REGION Network 49: Main Op Local Control
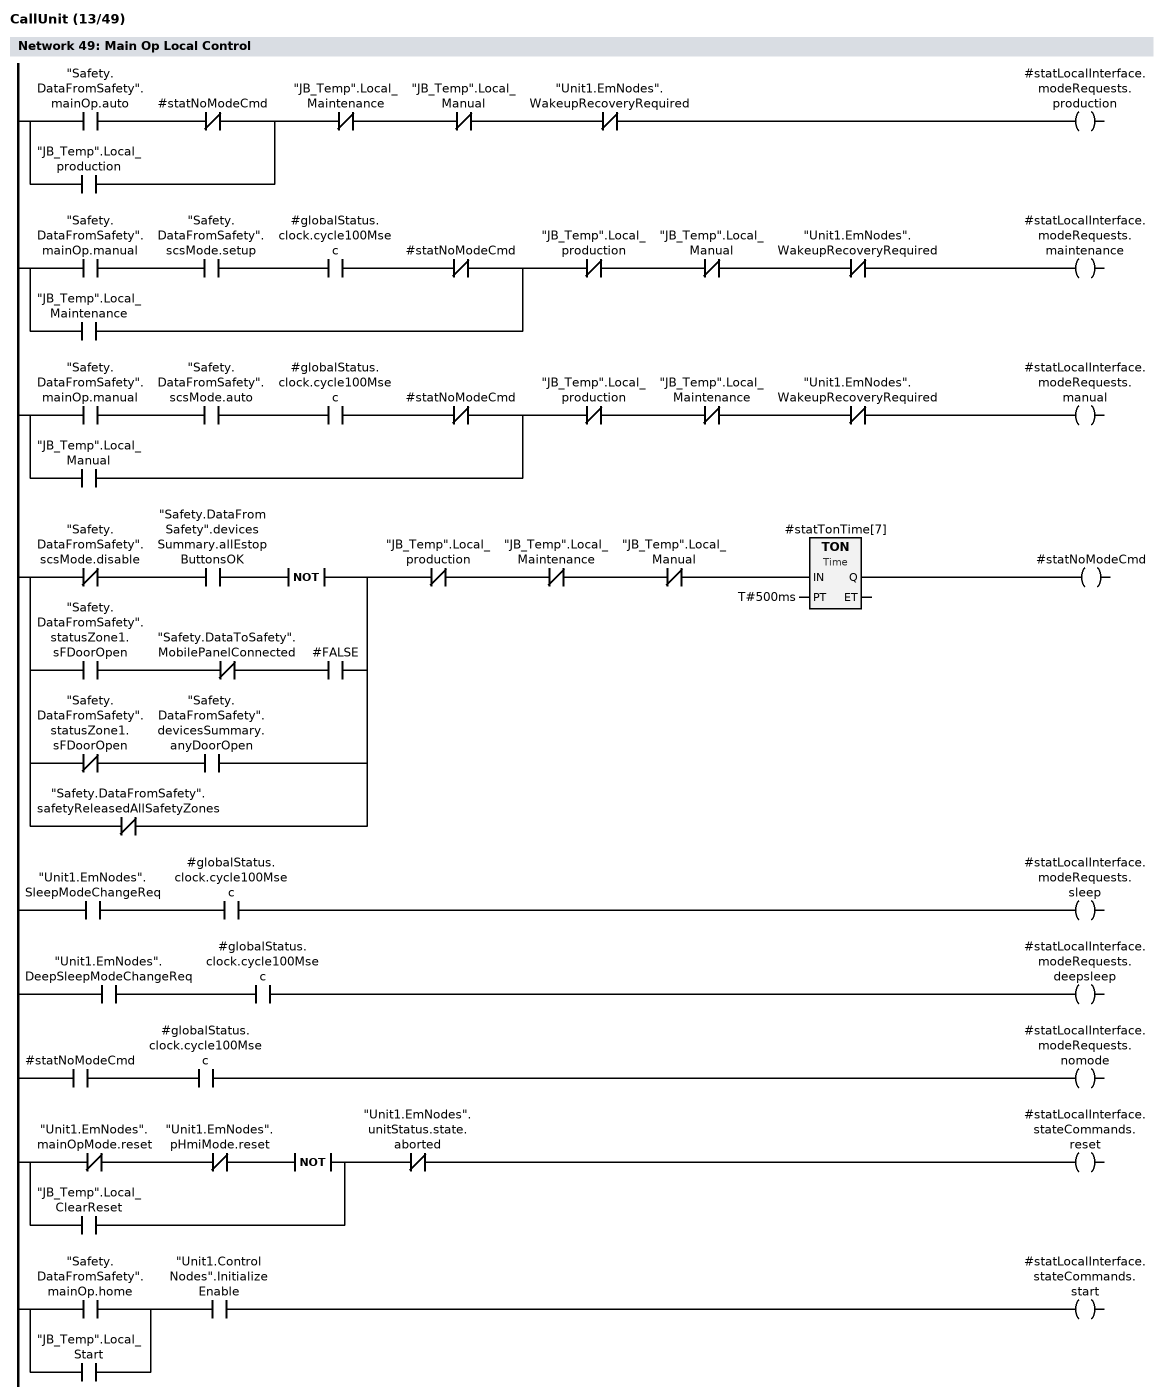
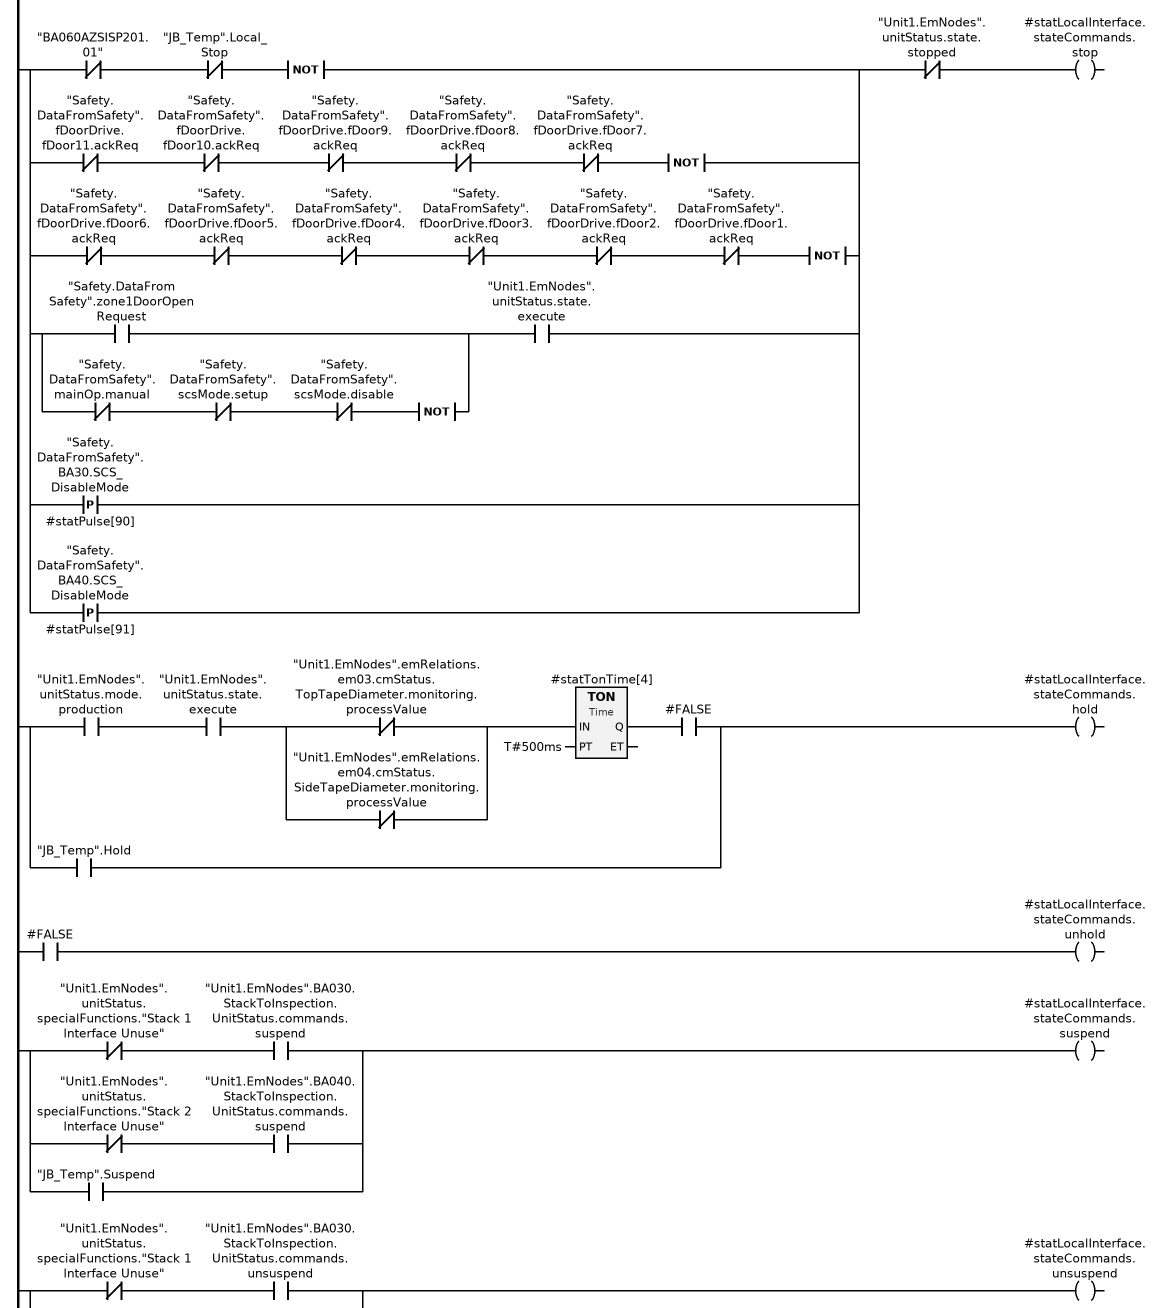
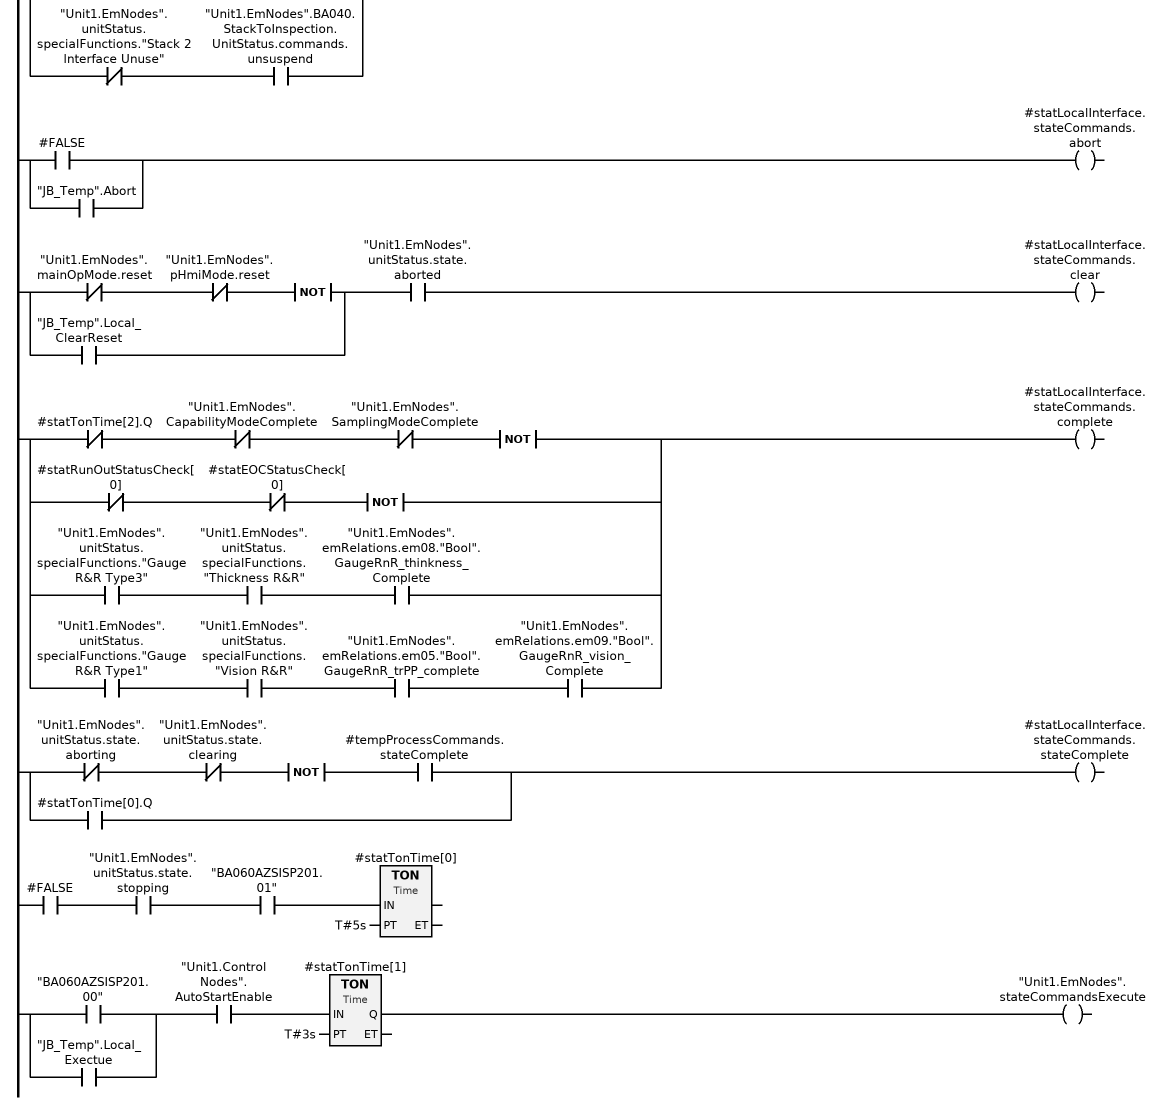
   RUNG wire#powerrail
      Contact( "Safety.DataFromSafety".mainOp.auto )
      I_Contact( #statNoModeCmd )
      wire#w1
      I_Contact( "JB_Temp".Local_Maintenance )
      I_Contact( "JB_Temp".Local_Manual )
      I_Contact( "Unit1.EmNodes".WakeupRecoveryRequired )
      Coil( #statLocalInterface.modeRequests.production )
   END_RUNG
   RUNG wire#powerrail
      Contact( "JB_Temp".Local_production )
   END_RUNG wire#w1
   RUNG wire#powerrail
      Contact( "Safety.DataFromSafety".mainOp.manual )
      Contact( "Safety.DataFromSafety".scsMode.setup )
      Contact( #globalStatus.clock.cycle100Msec )
      I_Contact( #statNoModeCmd )
      wire#w2
      I_Contact( "JB_Temp".Local_production )
      I_Contact( "JB_Temp".Local_Manual )
      I_Contact( "Unit1.EmNodes".WakeupRecoveryRequired )
      Coil( #statLocalInterface.modeRequests.maintenance )
   END_RUNG
   RUNG wire#powerrail
      Contact( "JB_Temp".Local_Maintenance )
   END_RUNG wire#w2
   RUNG wire#powerrail
      Contact( "Safety.DataFromSafety".mainOp.manual )
      Contact( "Safety.DataFromSafety".scsMode.auto )
      Contact( #globalStatus.clock.cycle100Msec )
      I_Contact( #statNoModeCmd )
      wire#w3
      I_Contact( "JB_Temp".Local_production )
      I_Contact( "JB_Temp".Local_Maintenance )
      I_Contact( "Unit1.EmNodes".WakeupRecoveryRequired )
      Coil( #statLocalInterface.modeRequests.manual )
   END_RUNG
   RUNG wire#powerrail
      Contact( "JB_Temp".Local_Manual )
   END_RUNG wire#w3
   RUNG wire#powerrail
      I_Contact( "Safety.DataFromSafety".scsMode.disable )
      Contact( "Safety.DataFromSafety".devicesSummary.allEstopButtonsOK )
      Not()
      wire#w4
      I_Contact( "JB_Temp".Local_production )
      I_Contact( "JB_Temp".Local_Maintenance )
      I_Contact( "JB_Temp".Local_Manual )
      { S7_Templates := "time_type := Time" } #statTonTime[7].TON(pt := T#500ms, et =>)
      Coil( #statNoModeCmd )
   END_RUNG
   RUNG wire#powerrail
      Contact( "Safety.DataFromSafety".statusZone1.sFDoorOpen )
      I_Contact( "Safety.DataToSafety".MobilePanelConnected )
      Contact( #FALSE )
   END_RUNG wire#w4
   RUNG wire#powerrail
      I_Contact( "Safety.DataFromSafety".statusZone1.sFDoorOpen )
      Contact( "Safety.DataFromSafety".devicesSummary.anyDoorOpen )
   END_RUNG wire#w4
   RUNG wire#powerrail
      I_Contact( "Safety.DataFromSafety".safetyReleasedAllSafetyZones )
   END_RUNG wire#w4
   RUNG wire#powerrail
      Contact( "Unit1.EmNodes".SleepModeChangeReq )
      Contact( #globalStatus.clock.cycle100Msec )
      Coil( #statLocalInterface.modeRequests.sleep )
   END_RUNG
   RUNG wire#powerrail
      Contact( "Unit1.EmNodes".DeepSleepModeChangeReq )
      Contact( #globalStatus.clock.cycle100Msec )
      Coil( #statLocalInterface.modeRequests.deepsleep )
   END_RUNG
   RUNG wire#powerrail
      Contact( #statNoModeCmd )
      Contact( #globalStatus.clock.cycle100Msec )
      Coil( #statLocalInterface.modeRequests.nomode )
   END_RUNG
   RUNG wire#powerrail
      I_Contact( "Unit1.EmNodes".mainOpMode.reset )
      I_Contact( "Unit1.EmNodes".pHmiMode.reset )
      Not()
      wire#w5
      I_Contact( "Unit1.EmNodes".unitStatus.state.aborted )
      Coil( #statLocalInterface.stateCommands.reset )
   END_RUNG
   RUNG wire#powerrail
      Contact( "JB_Temp".Local_ClearReset )
   END_RUNG wire#w5
   RUNG wire#powerrail
      Contact( "Safety.DataFromSafety".mainOp.home )
      wire#w6
      Contact( "Unit1.ControlNodes".InitializeEnable )
      Coil( #statLocalInterface.stateCommands.start )
   END_RUNG
   RUNG wire#powerrail
      Contact( "JB_Temp".Local_Start )
   END_RUNG wire#w6
   RUNG wire#powerrail
      I_Contact( "BA060AZSISP201.01" )
      I_Contact( "JB_Temp".Local_Stop )
      Not()
      wire#w7
      I_Contact( "Unit1.EmNodes".unitStatus.state.stopped )
      Coil( #statLocalInterface.stateCommands.stop )
   END_RUNG
   RUNG wire#powerrail
      I_Contact( "Safety.DataFromSafety".fDoorDrive.fDoor11.ackReq )
      I_Contact( "Safety.DataFromSafety".fDoorDrive.fDoor10.ackReq )
      I_Contact( "Safety.DataFromSafety".fDoorDrive.fDoor9.ackReq )
      I_Contact( "Safety.DataFromSafety".fDoorDrive.fDoor8.ackReq )
      I_Contact( "Safety.DataFromSafety".fDoorDrive.fDoor7.ackReq )
      Not()
   END_RUNG wire#w7
   RUNG wire#powerrail
      I_Contact( "Safety.DataFromSafety".fDoorDrive.fDoor6.ackReq )
      I_Contact( "Safety.DataFromSafety".fDoorDrive.fDoor5.ackReq )
      I_Contact( "Safety.DataFromSafety".fDoorDrive.fDoor4.ackReq )
      I_Contact( "Safety.DataFromSafety".fDoorDrive.fDoor3.ackReq )
      I_Contact( "Safety.DataFromSafety".fDoorDrive.fDoor2.ackReq )
      I_Contact( "Safety.DataFromSafety".fDoorDrive.fDoor1.ackReq )
      Not()
   END_RUNG wire#w7
   RUNG wire#powerrail
      Contact( "Safety.DataFromSafety".zone1DoorOpenRequest )
      wire#w8
      Contact( "Unit1.EmNodes".unitStatus.state.execute )
   END_RUNG wire#w7
   RUNG wire#powerrail
      I_Contact( "Safety.DataFromSafety".mainOp.manual )
      I_Contact( "Safety.DataFromSafety".scsMode.setup )
      I_Contact( "Safety.DataFromSafety".scsMode.disable )
      Not()
   END_RUNG wire#w8
   RUNG wire#powerrail
      P_Contact(operand := "Safety.DataFromSafety".BA30.SCS_DisableMode, bit := #statPulse[90])
   END_RUNG wire#w7
   RUNG wire#powerrail
      P_Contact(operand := "Safety.DataFromSafety".BA40.SCS_DisableMode, bit := #statPulse[91])
   END_RUNG wire#w7
   RUNG wire#powerrail
      Contact( "Unit1.EmNodes".unitStatus.mode.production )
      Contact( "Unit1.EmNodes".unitStatus.state.execute )
      wire#w9
      I_Contact( "Unit1.EmNodes".emRelations.em03.cmStatus.TopTapeDiameter.monitoring.processValue )
      wire#w10
      { S7_Templates := "time_type := Time" } #statTonTime[4].TON(pt := T#500ms, et =>)
      Contact( #FALSE )
      wire#w11
      Coil( #statLocalInterface.stateCommands.hold )
   END_RUNG
   RUNG wire#w9
      I_Contact( "Unit1.EmNodes".emRelations.em04.cmStatus.SideTapeDiameter.monitoring.processValue )
   END_RUNG wire#w10
   RUNG wire#powerrail
      Contact( "JB_Temp".Hold )
   END_RUNG wire#w11
   RUNG wire#powerrail
      Contact( #FALSE )
      Coil( #statLocalInterface.stateCommands.unhold )
   END_RUNG
   RUNG wire#powerrail
      I_Contact( "Unit1.EmNodes".unitStatus.specialFunctions."Stack 1 lnterface Unuse" )
      Contact( "Unit1.EmNodes".BA030.StackToInspection.UnitStatus.commands.suspend )
      wire#w12
      Coil( #statLocalInterface.stateCommands.suspend )
   END_RUNG
   RUNG wire#powerrail
      I_Contact( "Unit1.EmNodes".unitStatus.specialFunctions."Stack 2 lnterface Unuse" )
      Contact( "Unit1.EmNodes".BA040.StackToInspection.UnitStatus.commands.suspend )
   END_RUNG wire#w12
   RUNG wire#powerrail
      Contact( "JB_Temp".Suspend )
   END_RUNG wire#w12
   RUNG wire#powerrail
      I_Contact( "Unit1.EmNodes".unitStatus.specialFunctions."Stack 1 lnterface Unuse" )
      Contact( "Unit1.EmNodes".BA030.StackToInspection.UnitStatus.commands.unsuspend )
      wire#w13
      Coil( #statLocalInterface.stateCommands.unsuspend )
   END_RUNG
   RUNG wire#powerrail
      I_Contact( "Unit1.EmNodes".unitStatus.specialFunctions."Stack 2 lnterface Unuse" )
      Contact( "Unit1.EmNodes".BA040.StackToInspection.UnitStatus.commands.unsuspend )
   END_RUNG wire#w13
   RUNG wire#powerrail
      Contact( #FALSE )
      wire#w14
      Coil( #statLocalInterface.stateCommands.abort )
   END_RUNG
   RUNG wire#powerrail
      Contact( "JB_Temp".Abort )
   END_RUNG wire#w14
   RUNG wire#powerrail
      I_Contact( "Unit1.EmNodes".mainOpMode.reset )
      I_Contact( "Unit1.EmNodes".pHmiMode.reset )
      Not()
      wire#w15
      Contact( "Unit1.EmNodes".unitStatus.state.aborted )
      Coil( #statLocalInterface.stateCommands.clear )
   END_RUNG
   RUNG wire#powerrail
      Contact( "JB_Temp".Local_ClearReset )
   END_RUNG wire#w15
   RUNG wire#powerrail
      I_Contact( #statTonTime[2].Q )
      I_Contact( "Unit1.EmNodes".CapabilityModeComplete )
      I_Contact( "Unit1.EmNodes".SamplingModeComplete )
      Not()
      wire#w16
      Coil( #statLocalInterface.stateCommands.complete )
   END_RUNG
   RUNG wire#powerrail
      I_Contact( #statRunOutStatusCheck[0] )
      I_Contact( #statEOCStatusCheck[0] )
      Not()
   END_RUNG wire#w16
   RUNG wire#powerrail
      Contact( "Unit1.EmNodes".unitStatus.specialFunctions."Gauge R&R Type3" )
      Contact( "Unit1.EmNodes".unitStatus.specialFunctions."Thickness R&R" )
      Contact( "Unit1.EmNodes".emRelations.em08."Bool".GaugeRnR_thinkness_Complete )
   END_RUNG wire#w16
   RUNG wire#powerrail
      Contact( "Unit1.EmNodes".unitStatus.specialFunctions."Gauge R&R Type1" )
      Contact( "Unit1.EmNodes".unitStatus.specialFunctions."Vision R&R" )
      Contact( "Unit1.EmNodes".emRelations.em05."Bool".GaugeRnR_trPP_complete )
      Contact( "Unit1.EmNodes".emRelations.em09."Bool".GaugeRnR_vision_Complete )
   END_RUNG wire#w16
   RUNG wire#powerrail
      I_Contact( "Unit1.EmNodes".unitStatus.state.aborting )
      I_Contact( "Unit1.EmNodes".unitStatus.state.clearing )
      Not()
      Contact( #tempProcessCommands.stateComplete )
      wire#w17
      Coil( #statLocalInterface.stateCommands.stateComplete )
   END_RUNG
   RUNG wire#powerrail
      Contact( #statTonTime[0].Q )
   END_RUNG wire#w17
   RUNG wire#powerrail
      Contact( #FALSE )
      Contact( "Unit1.EmNodes".unitStatus.state.stopping )
      Contact( "BA060AZSISP201.01" )
      { S7_Templates := "time_type := Time" } #statTonTime[0].TON(pt := T#5s, et =>)
   END_RUNG
   RUNG wire#powerrail
      Contact( "BA060AZSISP201.00" )
      wire#w18
      Contact( "Unit1.ControlNodes".AutoStartEnable )
      { S7_Templates := "time_type := Time" } #statTonTime[1].TON(pt := T#3s, et =>)
      Coil( "Unit1.EmNodes".stateCommandsExecute )
   END_RUNG
   RUNG wire#powerrail
      Contact( "JB_Temp".Local_Exectue )
   END_RUNG wire#w18
   // the same network as SCL:
   #statLocalInterface.modeRequests.production := (("Safety.DataFromSafety".mainOp.auto AND NOT #statNoModeCmd) OR "JB_Temp".Local_production) AND NOT "JB_Temp".Local_Maintenance AND NOT "JB_Temp".Local_Manual AND NOT "Unit1.EmNodes".WakeupRecoveryRequired;
   #statLocalInterface.modeRequests.maintenance := (("Safety.DataFromSafety".mainOp.manual AND "Safety.DataFromSafety".scsMode.setup AND #globalStatus.clock.cycle100Msec AND NOT #statNoModeCmd) OR "JB_Temp".Local_Maintenance) AND NOT "JB_Temp".Local_production AND NOT "JB_Temp".Local_Manual AND NOT "Unit1.EmNodes".WakeupRecoveryRequired;
   #statLocalInterface.modeRequests.manual := (("Safety.DataFromSafety".mainOp.manual AND "Safety.DataFromSafety".scsMode.auto AND #globalStatus.clock.cycle100Msec AND NOT #statNoModeCmd) OR "JB_Temp".Local_Manual) AND NOT "JB_Temp".Local_production AND NOT "JB_Temp".Local_Maintenance AND NOT "Unit1.EmNodes".WakeupRecoveryRequired;
   #statTonTime[7].TON(IN := (NOT (NOT "Safety.DataFromSafety".scsMode.disable AND "Safety.DataFromSafety".devicesSummary.allEstopButtonsOK) OR ("Safety.DataFromSafety".statusZone1.sFDoorOpen AND NOT "Safety.DataToSafety".MobilePanelConnected AND #FALSE) OR (NOT "Safety.DataFromSafety".statusZone1.sFDoorOpen AND "Safety.DataFromSafety".devicesSummary.anyDoorOpen) OR NOT "Safety.DataFromSafety".safetyReleasedAllSafetyZones) AND NOT "JB_Temp".Local_production AND NOT "JB_Temp".Local_Maintenance AND NOT "JB_Temp".Local_Manual,
                       PT := T#500ms);
   #statNoModeCmd := #statTonTime[7].Q;
   #statLocalInterface.modeRequests.sleep := "Unit1.EmNodes".SleepModeChangeReq AND #globalStatus.clock.cycle100Msec;
   #statLocalInterface.modeRequests.deepsleep := "Unit1.EmNodes".DeepSleepModeChangeReq AND #globalStatus.clock.cycle100Msec;
   #statLocalInterface.modeRequests.nomode := #statNoModeCmd AND #globalStatus.clock.cycle100Msec;
   #statLocalInterface.stateCommands.reset := (NOT (NOT "Unit1.EmNodes".mainOpMode.reset AND NOT "Unit1.EmNodes".pHmiMode.reset) OR "JB_Temp".Local_ClearReset) AND NOT "Unit1.EmNodes".unitStatus.state.aborted;
   #statLocalInterface.stateCommands.start := ("Safety.DataFromSafety".mainOp.home OR "JB_Temp".Local_Start) AND "Unit1.ControlNodes".InitializeEnable;
   #_w1 := "Safety.DataFromSafety".BA30.SCS_DisableMode AND NOT #statPulse[90];   // rising edge of "Safety.DataFromSafety".BA30.SCS_DisableMode
   #statPulse[90] := "Safety.DataFromSafety".BA30.SCS_DisableMode;
   #_w2 := "Safety.DataFromSafety".BA40.SCS_DisableMode AND NOT #statPulse[91];   // rising edge of "Safety.DataFromSafety".BA40.SCS_DisableMode
   #statPulse[91] := "Safety.DataFromSafety".BA40.SCS_DisableMode;
   #statLocalInterface.stateCommands.stop := (NOT (NOT "BA060AZSISP201.01" AND NOT "JB_Temp".Local_Stop) OR NOT (NOT "Safety.DataFromSafety".fDoorDrive.fDoor11.ackReq AND NOT "Safety.DataFromSafety".fDoorDrive.fDoor10.ackReq AND NOT "Safety.DataFromSafety".fDoorDrive.fDoor9.ackReq AND NOT "Safety.DataFromSafety".fDoorDrive.fDoor8.ackReq AND NOT "Safety.DataFromSafety".fDoorDrive.fDoor7.ackReq) OR NOT (NOT "Safety.DataFromSafety".fDoorDrive.fDoor6.ackReq AND NOT "Safety.DataFromSafety".fDoorDrive.fDoor5.ackReq AND NOT "Safety.DataFromSafety".fDoorDrive.fDoor4.ackReq AND NOT "Safety.DataFromSafety".fDoorDrive.fDoor3.ackReq AND NOT "Safety.DataFromSafety".fDoorDrive.fDoor2.ackReq AND NOT "Safety.DataFromSafety".fDoorDrive.fDoor1.ackReq) OR (("Safety.DataFromSafety".zone1DoorOpenRequest OR NOT (NOT "Safety.DataFromSafety".mainOp.manual AND NOT "Safety.DataFromSafety".scsMode.setup AND NOT "Safety.DataFromSafety".scsMode.disable)) AND "Unit1.EmNodes".unitStatus.state.execute) OR #_w1 OR #_w2) AND NOT "Unit1.EmNodes".unitStatus.state.stopped;
   #statTonTime[4].TON(IN := "Unit1.EmNodes".unitStatus.mode.production AND "Unit1.EmNodes".unitStatus.state.execute AND (NOT "Unit1.EmNodes".emRelations.em03.cmStatus.TopTapeDiameter.monitoring.processValue OR NOT "Unit1.EmNodes".emRelations.em04.cmStatus.SideTapeDiameter.monitoring.processValue),
                       PT := T#500ms);
   #statLocalInterface.stateCommands.hold := (#statTonTime[4].Q AND #FALSE) OR "JB_Temp".Hold;
   #statLocalInterface.stateCommands.unhold := #FALSE;
   #statLocalInterface.stateCommands.suspend := (NOT "Unit1.EmNodes".unitStatus.specialFunctions."Stack 1 lnterface Unuse" AND "Unit1.EmNodes".BA030.StackToInspection.UnitStatus.commands.suspend) OR (NOT "Unit1.EmNodes".unitStatus.specialFunctions."Stack 2 lnterface Unuse" AND "Unit1.EmNodes".BA040.StackToInspection.UnitStatus.commands.suspend) OR "JB_Temp".Suspend;
   #statLocalInterface.stateCommands.unsuspend := (NOT "Unit1.EmNodes".unitStatus.specialFunctions."Stack 1 lnterface Unuse" AND "Unit1.EmNodes".BA030.StackToInspection.UnitStatus.commands.unsuspend) OR (NOT "Unit1.EmNodes".unitStatus.specialFunctions."Stack 2 lnterface Unuse" AND "Unit1.EmNodes".BA040.StackToInspection.UnitStatus.commands.unsuspend);
   #statLocalInterface.stateCommands.abort := #FALSE OR "JB_Temp".Abort;
   #statLocalInterface.stateCommands.clear := (NOT (NOT "Unit1.EmNodes".mainOpMode.reset AND NOT "Unit1.EmNodes".pHmiMode.reset) OR "JB_Temp".Local_ClearReset) AND "Unit1.EmNodes".unitStatus.state.aborted;
   #statLocalInterface.stateCommands.complete := NOT (NOT #statTonTime[2].Q AND NOT "Unit1.EmNodes".CapabilityModeComplete AND NOT "Unit1.EmNodes".SamplingModeComplete) OR NOT (NOT #statRunOutStatusCheck[0] AND NOT #statEOCStatusCheck[0]) OR ("Unit1.EmNodes".unitStatus.specialFunctions."Gauge R&R Type3" AND "Unit1.EmNodes".unitStatus.specialFunctions."Thickness R&R" AND "Unit1.EmNodes".emRelations.em08."Bool".GaugeRnR_thinkness_Complete) OR ("Unit1.EmNodes".unitStatus.specialFunctions."Gauge R&R Type1" AND "Unit1.EmNodes".unitStatus.specialFunctions."Vision R&R" AND "Unit1.EmNodes".emRelations.em05."Bool".GaugeRnR_trPP_complete AND "Unit1.EmNodes".emRelations.em09."Bool".GaugeRnR_vision_Complete);
   #statLocalInterface.stateCommands.stateComplete := (NOT (NOT "Unit1.EmNodes".unitStatus.state.aborting AND NOT "Unit1.EmNodes".unitStatus.state.clearing) AND #tempProcessCommands.stateComplete) OR #statTonTime[0].Q;
   #statTonTime[0].TON(IN := #FALSE AND "Unit1.EmNodes".unitStatus.state.stopping AND "BA060AZSISP201.01",
                       PT := T#5s);
   #statTonTime[1].TON(IN := ("BA060AZSISP201.00" OR "JB_Temp".Local_Exectue) AND "Unit1.ControlNodes".AutoStartEnable,
                       PT := T#3s);
   "Unit1.EmNodes".stateCommandsExecute := #statTonTime[1].Q;
END_REGION

REGION Network 50: Main Op Lamp
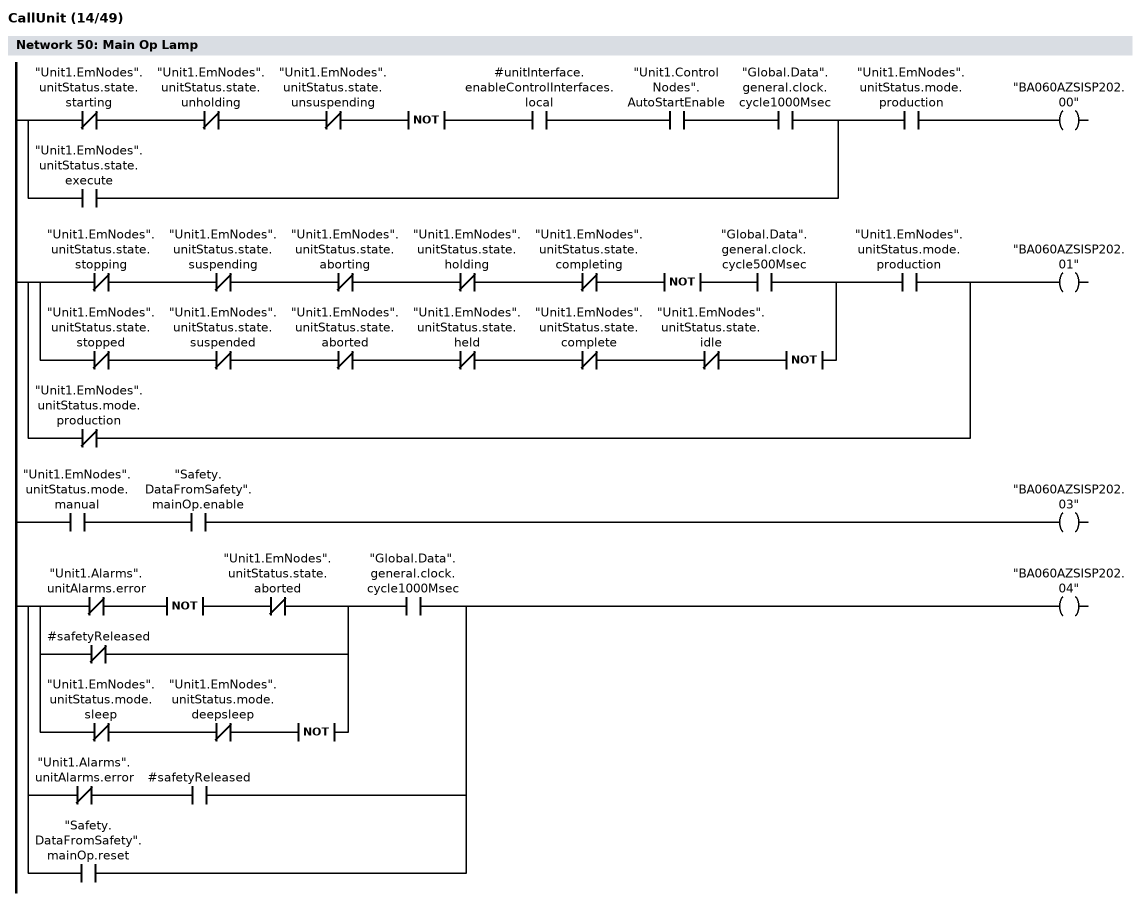
   RUNG wire#powerrail
      I_Contact( "Unit1.EmNodes".unitStatus.state.starting )
      I_Contact( "Unit1.EmNodes".unitStatus.state.unholding )
      I_Contact( "Unit1.EmNodes".unitStatus.state.unsuspending )
      Not()
      Contact( #unitInterface.enableControlInterfaces.local )
      Contact( "Unit1.ControlNodes".AutoStartEnable )
      Contact( "Global.Data".general.clock.cycle1000Msec )
      wire#w1
      Contact( "Unit1.EmNodes".unitStatus.mode.production )
      Coil( "BA060AZSISP202.00" )
   END_RUNG
   RUNG wire#powerrail
      Contact( "Unit1.EmNodes".unitStatus.state.execute )
   END_RUNG wire#w1
   RUNG wire#powerrail
      I_Contact( "Unit1.EmNodes".unitStatus.state.stopping )
      I_Contact( "Unit1.EmNodes".unitStatus.state.suspending )
      I_Contact( "Unit1.EmNodes".unitStatus.state.aborting )
      I_Contact( "Unit1.EmNodes".unitStatus.state.holding )
      I_Contact( "Unit1.EmNodes".unitStatus.state.completing )
      Not()
      Contact( "Global.Data".general.clock.cycle500Msec )
      wire#w2
      Contact( "Unit1.EmNodes".unitStatus.mode.production )
      wire#w3
      Coil( "BA060AZSISP202.01" )
   END_RUNG
   RUNG wire#powerrail
      I_Contact( "Unit1.EmNodes".unitStatus.state.stopped )
      I_Contact( "Unit1.EmNodes".unitStatus.state.suspended )
      I_Contact( "Unit1.EmNodes".unitStatus.state.aborted )
      I_Contact( "Unit1.EmNodes".unitStatus.state.held )
      I_Contact( "Unit1.EmNodes".unitStatus.state.complete )
      I_Contact( "Unit1.EmNodes".unitStatus.state.idle )
      Not()
   END_RUNG wire#w2
   RUNG wire#powerrail
      I_Contact( "Unit1.EmNodes".unitStatus.mode.production )
   END_RUNG wire#w3
   RUNG wire#powerrail
      Contact( "Unit1.EmNodes".unitStatus.mode.manual )
      Contact( "Safety.DataFromSafety".mainOp.enable )
      Coil( "BA060AZSISP202.03" )
   END_RUNG
   RUNG wire#powerrail
      I_Contact( "Unit1.Alarms".unitAlarms.error )
      Not()
      I_Contact( "Unit1.EmNodes".unitStatus.state.aborted )
      wire#w4
      Contact( "Global.Data".general.clock.cycle1000Msec )
      wire#w5
      Coil( "BA060AZSISP202.04" )
   END_RUNG
   RUNG wire#powerrail
      I_Contact( #safetyReleased )
   END_RUNG wire#w4
   RUNG wire#powerrail
      I_Contact( "Unit1.EmNodes".unitStatus.mode.sleep )
      I_Contact( "Unit1.EmNodes".unitStatus.mode.deepsleep )
      Not()
   END_RUNG wire#w4
   RUNG wire#powerrail
      I_Contact( "Unit1.Alarms".unitAlarms.error )
      Contact( #safetyReleased )
   END_RUNG wire#w5
   RUNG wire#powerrail
      Contact( "Safety.DataFromSafety".mainOp.reset )
   END_RUNG wire#w5
   // the same network as SCL:
   "BA060AZSISP202.00" := ((NOT (NOT "Unit1.EmNodes".unitStatus.state.starting AND NOT "Unit1.EmNodes".unitStatus.state.unholding AND NOT "Unit1.EmNodes".unitStatus.state.unsuspending) AND #unitInterface.enableControlInterfaces.local AND "Unit1.ControlNodes".AutoStartEnable AND "Global.Data".general.clock.cycle1000Msec) OR "Unit1.EmNodes".unitStatus.state.execute) AND "Unit1.EmNodes".unitStatus.mode.production;
   "BA060AZSISP202.01" := (((NOT (NOT "Unit1.EmNodes".unitStatus.state.stopping AND NOT "Unit1.EmNodes".unitStatus.state.suspending AND NOT "Unit1.EmNodes".unitStatus.state.aborting AND NOT "Unit1.EmNodes".unitStatus.state.holding AND NOT "Unit1.EmNodes".unitStatus.state.completing) AND "Global.Data".general.clock.cycle500Msec) OR NOT (NOT "Unit1.EmNodes".unitStatus.state.stopped AND NOT "Unit1.EmNodes".unitStatus.state.suspended AND NOT "Unit1.EmNodes".unitStatus.state.aborted AND NOT "Unit1.EmNodes".unitStatus.state.held AND NOT "Unit1.EmNodes".unitStatus.state.complete AND NOT "Unit1.EmNodes".unitStatus.state.idle)) AND "Unit1.EmNodes".unitStatus.mode.production) OR NOT "Unit1.EmNodes".unitStatus.mode.production;
   "BA060AZSISP202.03" := "Unit1.EmNodes".unitStatus.mode.manual AND "Safety.DataFromSafety".mainOp.enable;
   "BA060AZSISP202.04" := (((NOT (NOT "Unit1.Alarms".unitAlarms.error) AND NOT "Unit1.EmNodes".unitStatus.state.aborted) OR NOT #safetyReleased OR NOT (NOT "Unit1.EmNodes".unitStatus.mode.sleep AND NOT "Unit1.EmNodes".unitStatus.mode.deepsleep)) AND "Global.Data".general.clock.cycle1000Msec) OR (NOT "Unit1.Alarms".unitAlarms.error AND #safetyReleased) OR "Safety.DataFromSafety".mainOp.reset;
END_REGION

REGION Network 51: ******************** Data To Safety Mapping ********************
END_REGION

REGION Network 52: Unit Mode
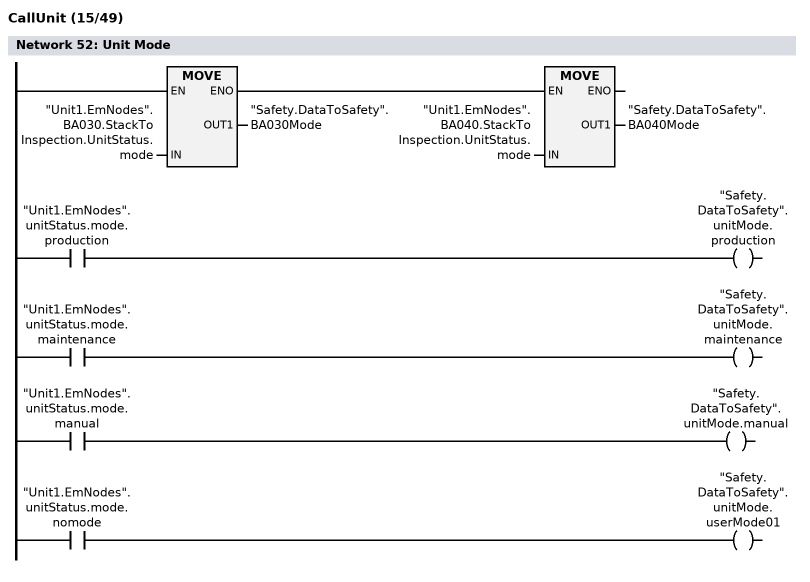
   RUNG wire#powerrail
      Move(in := "Unit1.EmNodes".BA030.StackToInspection.UnitStatus.mode, out1 => "Safety.DataToSafety".BA030Mode)
      Move(in := "Unit1.EmNodes".BA040.StackToInspection.UnitStatus.mode, out1 => "Safety.DataToSafety".BA040Mode)
   END_RUNG
   RUNG wire#powerrail
      Contact( "Unit1.EmNodes".unitStatus.mode.production )
      Coil( "Safety.DataToSafety".unitMode.production )
   END_RUNG
   RUNG wire#powerrail
      Contact( "Unit1.EmNodes".unitStatus.mode.maintenance )
      Coil( "Safety.DataToSafety".unitMode.maintenance )
   END_RUNG
   RUNG wire#powerrail
      Contact( "Unit1.EmNodes".unitStatus.mode.manual )
      Coil( "Safety.DataToSafety".unitMode.manual )
   END_RUNG
   RUNG wire#powerrail
      Contact( "Unit1.EmNodes".unitStatus.mode.nomode )
      Coil( "Safety.DataToSafety".unitMode.userMode01 )
   END_RUNG
   // the same network as SCL:
   "Safety.DataToSafety".BA030Mode := "Unit1.EmNodes".BA030.StackToInspection.UnitStatus.mode;
   "Safety.DataToSafety".BA040Mode := "Unit1.EmNodes".BA040.StackToInspection.UnitStatus.mode;
   "Safety.DataToSafety".unitMode.production := "Unit1.EmNodes".unitStatus.mode.production;
   "Safety.DataToSafety".unitMode.maintenance := "Unit1.EmNodes".unitStatus.mode.maintenance;
   "Safety.DataToSafety".unitMode.manual := "Unit1.EmNodes".unitStatus.mode.manual;
   "Safety.DataToSafety".unitMode.userMode01 := "Unit1.EmNodes".unitStatus.mode.nomode;
END_REGION

REGION Network 53: Unit States
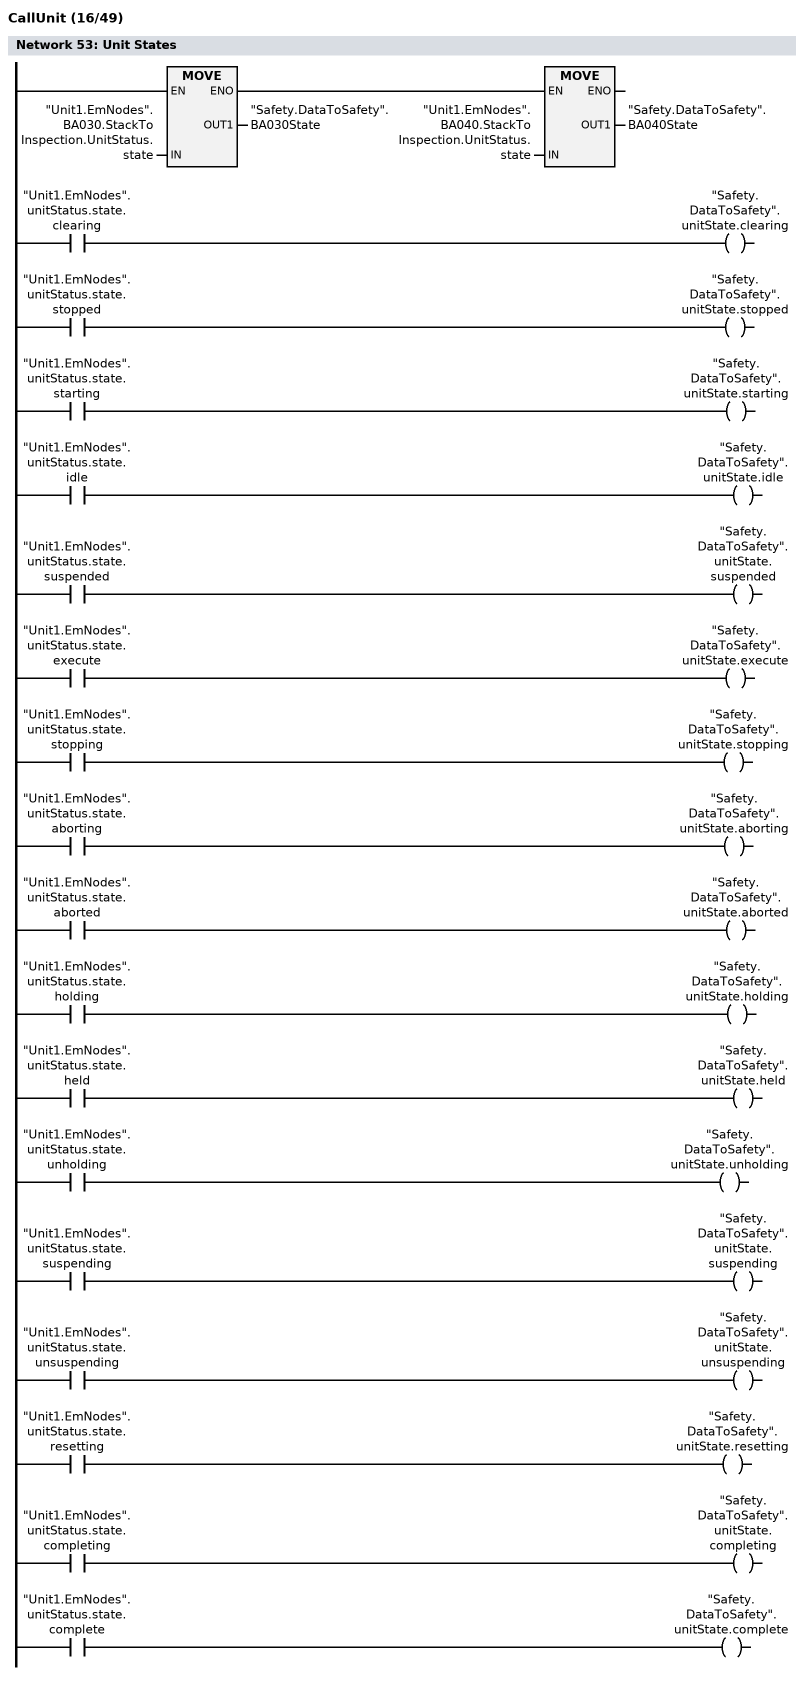
   RUNG wire#powerrail
      Move(in := "Unit1.EmNodes".BA030.StackToInspection.UnitStatus.state, out1 => "Safety.DataToSafety".BA030State)
      Move(in := "Unit1.EmNodes".BA040.StackToInspection.UnitStatus.state, out1 => "Safety.DataToSafety".BA040State)
   END_RUNG
   RUNG wire#powerrail
      Contact( "Unit1.EmNodes".unitStatus.state.clearing )
      Coil( "Safety.DataToSafety".unitState.clearing )
   END_RUNG
   RUNG wire#powerrail
      Contact( "Unit1.EmNodes".unitStatus.state.stopped )
      Coil( "Safety.DataToSafety".unitState.stopped )
   END_RUNG
   RUNG wire#powerrail
      Contact( "Unit1.EmNodes".unitStatus.state.starting )
      Coil( "Safety.DataToSafety".unitState.starting )
   END_RUNG
   RUNG wire#powerrail
      Contact( "Unit1.EmNodes".unitStatus.state.idle )
      Coil( "Safety.DataToSafety".unitState.idle )
   END_RUNG
   RUNG wire#powerrail
      Contact( "Unit1.EmNodes".unitStatus.state.suspended )
      Coil( "Safety.DataToSafety".unitState.suspended )
   END_RUNG
   RUNG wire#powerrail
      Contact( "Unit1.EmNodes".unitStatus.state.execute )
      Coil( "Safety.DataToSafety".unitState.execute )
   END_RUNG
   RUNG wire#powerrail
      Contact( "Unit1.EmNodes".unitStatus.state.stopping )
      Coil( "Safety.DataToSafety".unitState.stopping )
   END_RUNG
   RUNG wire#powerrail
      Contact( "Unit1.EmNodes".unitStatus.state.aborting )
      Coil( "Safety.DataToSafety".unitState.aborting )
   END_RUNG
   RUNG wire#powerrail
      Contact( "Unit1.EmNodes".unitStatus.state.aborted )
      Coil( "Safety.DataToSafety".unitState.aborted )
   END_RUNG
   RUNG wire#powerrail
      Contact( "Unit1.EmNodes".unitStatus.state.holding )
      Coil( "Safety.DataToSafety".unitState.holding )
   END_RUNG
   RUNG wire#powerrail
      Contact( "Unit1.EmNodes".unitStatus.state.held )
      Coil( "Safety.DataToSafety".unitState.held )
   END_RUNG
   RUNG wire#powerrail
      Contact( "Unit1.EmNodes".unitStatus.state.unholding )
      Coil( "Safety.DataToSafety".unitState.unholding )
   END_RUNG
   RUNG wire#powerrail
      Contact( "Unit1.EmNodes".unitStatus.state.suspending )
      Coil( "Safety.DataToSafety".unitState.suspending )
   END_RUNG
   RUNG wire#powerrail
      Contact( "Unit1.EmNodes".unitStatus.state.unsuspending )
      Coil( "Safety.DataToSafety".unitState.unsuspending )
   END_RUNG
   RUNG wire#powerrail
      Contact( "Unit1.EmNodes".unitStatus.state.resetting )
      Coil( "Safety.DataToSafety".unitState.resetting )
   END_RUNG
   RUNG wire#powerrail
      Contact( "Unit1.EmNodes".unitStatus.state.completing )
      Coil( "Safety.DataToSafety".unitState.completing )
   END_RUNG
   RUNG wire#powerrail
      Contact( "Unit1.EmNodes".unitStatus.state.complete )
      Coil( "Safety.DataToSafety".unitState.complete )
   END_RUNG
   // the same network as SCL:
   "Safety.DataToSafety".BA030State := "Unit1.EmNodes".BA030.StackToInspection.UnitStatus.state;
   "Safety.DataToSafety".BA040State := "Unit1.EmNodes".BA040.StackToInspection.UnitStatus.state;
   "Safety.DataToSafety".unitState.clearing := "Unit1.EmNodes".unitStatus.state.clearing;
   "Safety.DataToSafety".unitState.stopped := "Unit1.EmNodes".unitStatus.state.stopped;
   "Safety.DataToSafety".unitState.starting := "Unit1.EmNodes".unitStatus.state.starting;
   "Safety.DataToSafety".unitState.idle := "Unit1.EmNodes".unitStatus.state.idle;
   "Safety.DataToSafety".unitState.suspended := "Unit1.EmNodes".unitStatus.state.suspended;
   "Safety.DataToSafety".unitState.execute := "Unit1.EmNodes".unitStatus.state.execute;
   "Safety.DataToSafety".unitState.stopping := "Unit1.EmNodes".unitStatus.state.stopping;
   "Safety.DataToSafety".unitState.aborting := "Unit1.EmNodes".unitStatus.state.aborting;
   "Safety.DataToSafety".unitState.aborted := "Unit1.EmNodes".unitStatus.state.aborted;
   "Safety.DataToSafety".unitState.holding := "Unit1.EmNodes".unitStatus.state.holding;
   "Safety.DataToSafety".unitState.held := "Unit1.EmNodes".unitStatus.state.held;
   "Safety.DataToSafety".unitState.unholding := "Unit1.EmNodes".unitStatus.state.unholding;
   "Safety.DataToSafety".unitState.suspending := "Unit1.EmNodes".unitStatus.state.suspending;
   "Safety.DataToSafety".unitState.unsuspending := "Unit1.EmNodes".unitStatus.state.unsuspending;
   "Safety.DataToSafety".unitState.resetting := "Unit1.EmNodes".unitStatus.state.resetting;
   "Safety.DataToSafety".unitState.completing := "Unit1.EmNodes".unitStatus.state.completing;
   "Safety.DataToSafety".unitState.complete := "Unit1.EmNodes".unitStatus.state.complete;
END_REGION

REGION Network 54: Deselect BA30, BA40
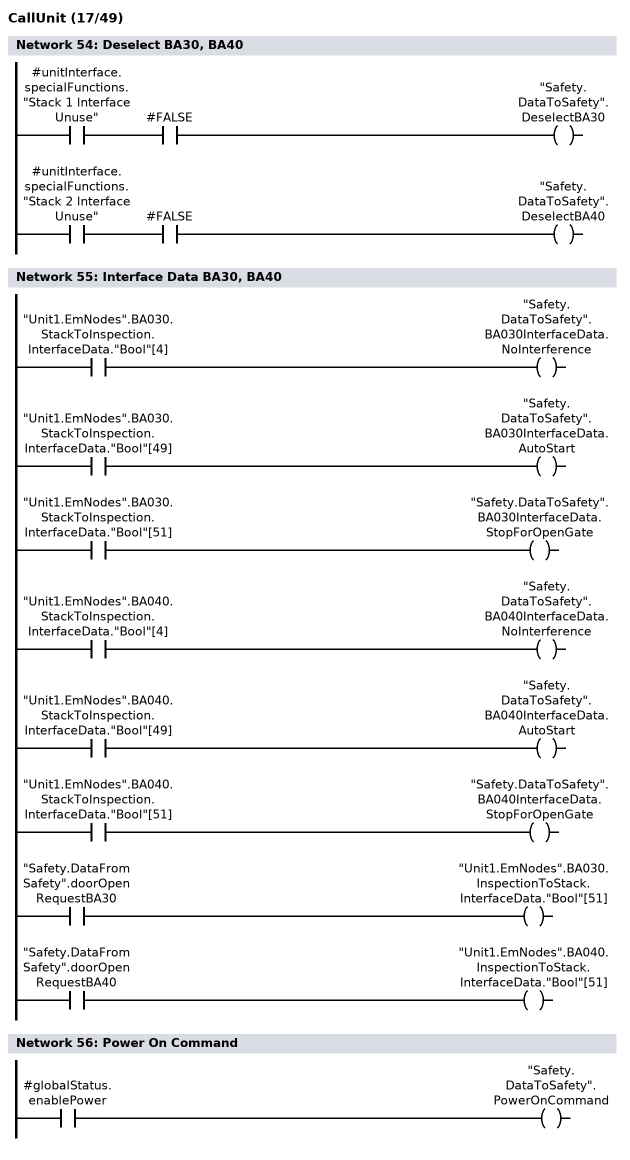
   RUNG wire#powerrail
      Contact( #unitInterface.specialFunctions."Stack 1 lnterface Unuse" )
      Contact( #FALSE )
      Coil( "Safety.DataToSafety".DeselectBA30 )
   END_RUNG
   RUNG wire#powerrail
      Contact( #unitInterface.specialFunctions."Stack 2 lnterface Unuse" )
      Contact( #FALSE )
      Coil( "Safety.DataToSafety".DeselectBA40 )
   END_RUNG
   // the same network as SCL:
   "Safety.DataToSafety".DeselectBA30 := #unitInterface.specialFunctions."Stack 1 lnterface Unuse" AND #FALSE;
   "Safety.DataToSafety".DeselectBA40 := #unitInterface.specialFunctions."Stack 2 lnterface Unuse" AND #FALSE;
END_REGION

REGION Network 55: Interface Data BA30, BA40
   RUNG wire#powerrail
      Contact( "Unit1.EmNodes".BA030.StackToInspection.InterfaceData."Bool"[4] )
      Coil( "Safety.DataToSafety".BA030InterfaceData.NoInterference )
   END_RUNG
   RUNG wire#powerrail
      Contact( "Unit1.EmNodes".BA030.StackToInspection.InterfaceData."Bool"[49] )
      Coil( "Safety.DataToSafety".BA030InterfaceData.AutoStart )
   END_RUNG
   RUNG wire#powerrail
      Contact( "Unit1.EmNodes".BA030.StackToInspection.InterfaceData."Bool"[51] )
      Coil( "Safety.DataToSafety".BA030InterfaceData.StopForOpenGate )
   END_RUNG
   RUNG wire#powerrail
      Contact( "Unit1.EmNodes".BA040.StackToInspection.InterfaceData."Bool"[4] )
      Coil( "Safety.DataToSafety".BA040InterfaceData.NoInterference )
   END_RUNG
   RUNG wire#powerrail
      Contact( "Unit1.EmNodes".BA040.StackToInspection.InterfaceData."Bool"[49] )
      Coil( "Safety.DataToSafety".BA040InterfaceData.AutoStart )
   END_RUNG
   RUNG wire#powerrail
      Contact( "Unit1.EmNodes".BA040.StackToInspection.InterfaceData."Bool"[51] )
      Coil( "Safety.DataToSafety".BA040InterfaceData.StopForOpenGate )
   END_RUNG
   RUNG wire#powerrail
      Contact( "Safety.DataFromSafety".doorOpenRequestBA30 )
      Coil( "Unit1.EmNodes".BA030.InspectionToStack.InterfaceData."Bool"[51] )
   END_RUNG
   RUNG wire#powerrail
      Contact( "Safety.DataFromSafety".doorOpenRequestBA40 )
      Coil( "Unit1.EmNodes".BA040.InspectionToStack.InterfaceData."Bool"[51] )
   END_RUNG
   // the same network as SCL:
   "Safety.DataToSafety".BA030InterfaceData.NoInterference := "Unit1.EmNodes".BA030.StackToInspection.InterfaceData."Bool"[4];
   "Safety.DataToSafety".BA030InterfaceData.AutoStart := "Unit1.EmNodes".BA030.StackToInspection.InterfaceData."Bool"[49];
   "Safety.DataToSafety".BA030InterfaceData.StopForOpenGate := "Unit1.EmNodes".BA030.StackToInspection.InterfaceData."Bool"[51];
   "Safety.DataToSafety".BA040InterfaceData.NoInterference := "Unit1.EmNodes".BA040.StackToInspection.InterfaceData."Bool"[4];
   "Safety.DataToSafety".BA040InterfaceData.AutoStart := "Unit1.EmNodes".BA040.StackToInspection.InterfaceData."Bool"[49];
   "Safety.DataToSafety".BA040InterfaceData.StopForOpenGate := "Unit1.EmNodes".BA040.StackToInspection.InterfaceData."Bool"[51];
   "Unit1.EmNodes".BA030.InspectionToStack.InterfaceData."Bool"[51] := "Safety.DataFromSafety".doorOpenRequestBA30;
   "Unit1.EmNodes".BA040.InspectionToStack.InterfaceData."Bool"[51] := "Safety.DataFromSafety".doorOpenRequestBA40;
END_REGION

REGION Network 56: Power On Command
   RUNG wire#powerrail
      Contact( #globalStatus.enablePower )
      Coil( "Safety.DataToSafety".PowerOnCommand )
   END_RUNG
   // the same network as SCL:
   "Safety.DataToSafety".PowerOnCommand := #globalStatus.enablePower;
END_REGION

REGION Network 57: OP Lamp
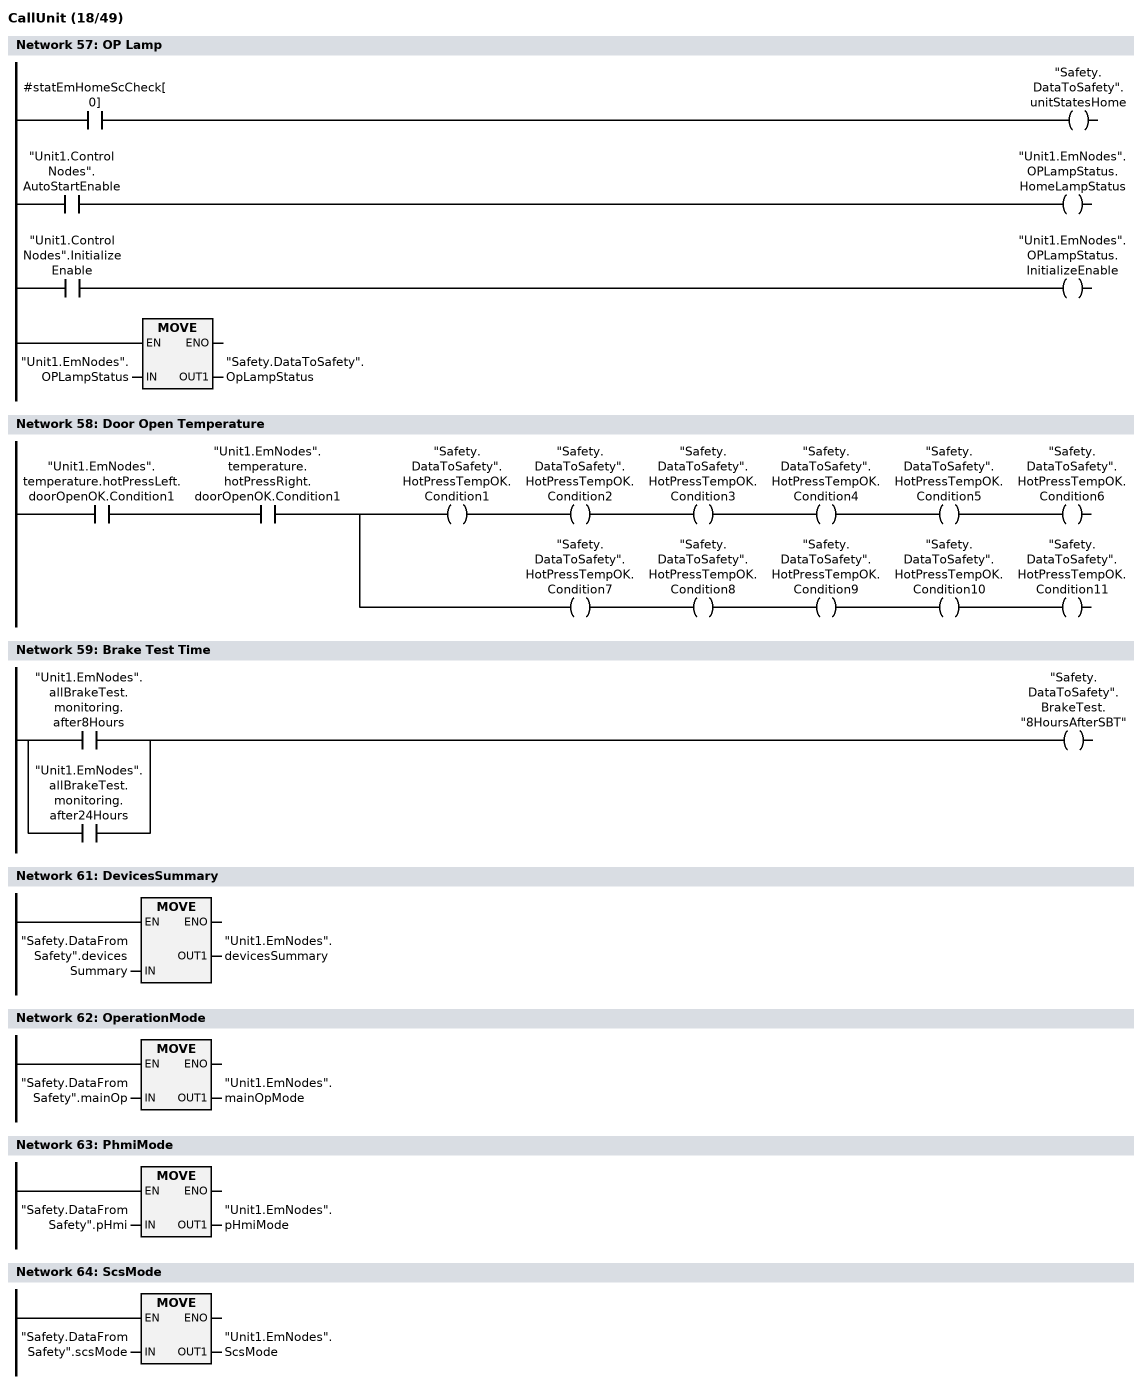
   RUNG wire#powerrail
      Contact( #statEmHomeScCheck[0] )
      Coil( "Safety.DataToSafety".unitStatesHome )
   END_RUNG
   RUNG wire#powerrail
      Contact( "Unit1.ControlNodes".AutoStartEnable )
      Coil( "Unit1.EmNodes".OPLampStatus.HomeLampStatus )
   END_RUNG
   RUNG wire#powerrail
      Contact( "Unit1.ControlNodes".InitializeEnable )
      Coil( "Unit1.EmNodes".OPLampStatus.InitializeEnable )
   END_RUNG
   RUNG wire#powerrail
      Move(in := "Unit1.EmNodes".OPLampStatus, out1 => "Safety.DataToSafety".OpLampStatus)
   END_RUNG
   // the same network as SCL:
   "Safety.DataToSafety".unitStatesHome := #statEmHomeScCheck[0];
   "Unit1.EmNodes".OPLampStatus.HomeLampStatus := "Unit1.ControlNodes".AutoStartEnable;
   "Unit1.EmNodes".OPLampStatus.InitializeEnable := "Unit1.ControlNodes".InitializeEnable;
   "Safety.DataToSafety".OpLampStatus := "Unit1.EmNodes".OPLampStatus;
END_REGION

REGION Network 58: Door Open Temperature
   RUNG wire#powerrail
      Contact( "Unit1.EmNodes".temperature.hotPressLeft.doorOpenOK.Condition1 )
      Contact( "Unit1.EmNodes".temperature.hotPressRight.doorOpenOK.Condition1 )
      wire#w1
      Coil( "Safety.DataToSafety".HotPressTempOK.Condition1 )
      Coil( "Safety.DataToSafety".HotPressTempOK.Condition2 )
      Coil( "Safety.DataToSafety".HotPressTempOK.Condition3 )
      Coil( "Safety.DataToSafety".HotPressTempOK.Condition4 )
      Coil( "Safety.DataToSafety".HotPressTempOK.Condition5 )
      Coil( "Safety.DataToSafety".HotPressTempOK.Condition6 )
   END_RUNG
   RUNG wire#w1
      Coil( "Safety.DataToSafety".HotPressTempOK.Condition7 )
      Coil( "Safety.DataToSafety".HotPressTempOK.Condition8 )
      Coil( "Safety.DataToSafety".HotPressTempOK.Condition9 )
      Coil( "Safety.DataToSafety".HotPressTempOK.Condition10 )
      Coil( "Safety.DataToSafety".HotPressTempOK.Condition11 )
   END_RUNG
   // the same network as SCL:
   "Safety.DataToSafety".HotPressTempOK.Condition1 := "Unit1.EmNodes".temperature.hotPressLeft.doorOpenOK.Condition1 AND "Unit1.EmNodes".temperature.hotPressRight.doorOpenOK.Condition1;
   "Safety.DataToSafety".HotPressTempOK.Condition2 := "Safety.DataToSafety".HotPressTempOK.Condition1;
   "Safety.DataToSafety".HotPressTempOK.Condition3 := "Safety.DataToSafety".HotPressTempOK.Condition1;
   "Safety.DataToSafety".HotPressTempOK.Condition4 := "Safety.DataToSafety".HotPressTempOK.Condition1;
   "Safety.DataToSafety".HotPressTempOK.Condition5 := "Safety.DataToSafety".HotPressTempOK.Condition1;
   "Safety.DataToSafety".HotPressTempOK.Condition6 := "Safety.DataToSafety".HotPressTempOK.Condition1;
   "Safety.DataToSafety".HotPressTempOK.Condition7 := "Safety.DataToSafety".HotPressTempOK.Condition1;
   "Safety.DataToSafety".HotPressTempOK.Condition8 := "Safety.DataToSafety".HotPressTempOK.Condition1;
   "Safety.DataToSafety".HotPressTempOK.Condition9 := "Safety.DataToSafety".HotPressTempOK.Condition1;
   "Safety.DataToSafety".HotPressTempOK.Condition10 := "Safety.DataToSafety".HotPressTempOK.Condition1;
   "Safety.DataToSafety".HotPressTempOK.Condition11 := "Safety.DataToSafety".HotPressTempOK.Condition1;
END_REGION

REGION Network 59: Brake Test Time
   RUNG wire#powerrail
      Contact( "Unit1.EmNodes".allBrakeTest.monitoring.after8Hours )
      wire#w1
      Coil( "Safety.DataToSafety".BrakeTest."8HoursAfterSBT" )
   END_RUNG
   RUNG wire#powerrail
      Contact( "Unit1.EmNodes".allBrakeTest.monitoring.after24Hours )
   END_RUNG wire#w1
   // the same network as SCL:
   "Safety.DataToSafety".BrakeTest."8HoursAfterSBT" := "Unit1.EmNodes".allBrakeTest.monitoring.after8Hours OR "Unit1.EmNodes".allBrakeTest.monitoring.after24Hours;
END_REGION

REGION Network 60: ******************** Data From Safety Mapping ********************
END_REGION

REGION Network 61: DevicesSummary
   RUNG wire#powerrail
      Move(in := "Safety.DataFromSafety".devicesSummary, out1 => "Unit1.EmNodes".devicesSummary)
   END_RUNG
   // the same network as SCL:
   "Unit1.EmNodes".devicesSummary := "Safety.DataFromSafety".devicesSummary;
END_REGION

REGION Network 62: OperationMode
   RUNG wire#powerrail
      Move(in := "Safety.DataFromSafety".mainOp, out1 => "Unit1.EmNodes".mainOpMode)
   END_RUNG
   // the same network as SCL:
   "Unit1.EmNodes".mainOpMode := "Safety.DataFromSafety".mainOp;
END_REGION

REGION Network 63: PhmiMode
   RUNG wire#powerrail
      Move(in := "Safety.DataFromSafety".pHmi, out1 => "Unit1.EmNodes".pHmiMode)
   END_RUNG
   // the same network as SCL:
   "Unit1.EmNodes".pHmiMode := "Safety.DataFromSafety".pHmi;
END_REGION

REGION Network 64: ScsMode
   RUNG wire#powerrail
      Move(in := "Safety.DataFromSafety".scsMode, out1 => "Unit1.EmNodes".ScsMode)
   END_RUNG
   // the same network as SCL:
   "Unit1.EmNodes".ScsMode := "Safety.DataFromSafety".scsMode;
END_REGION

REGION Network 65: ScrapBox1
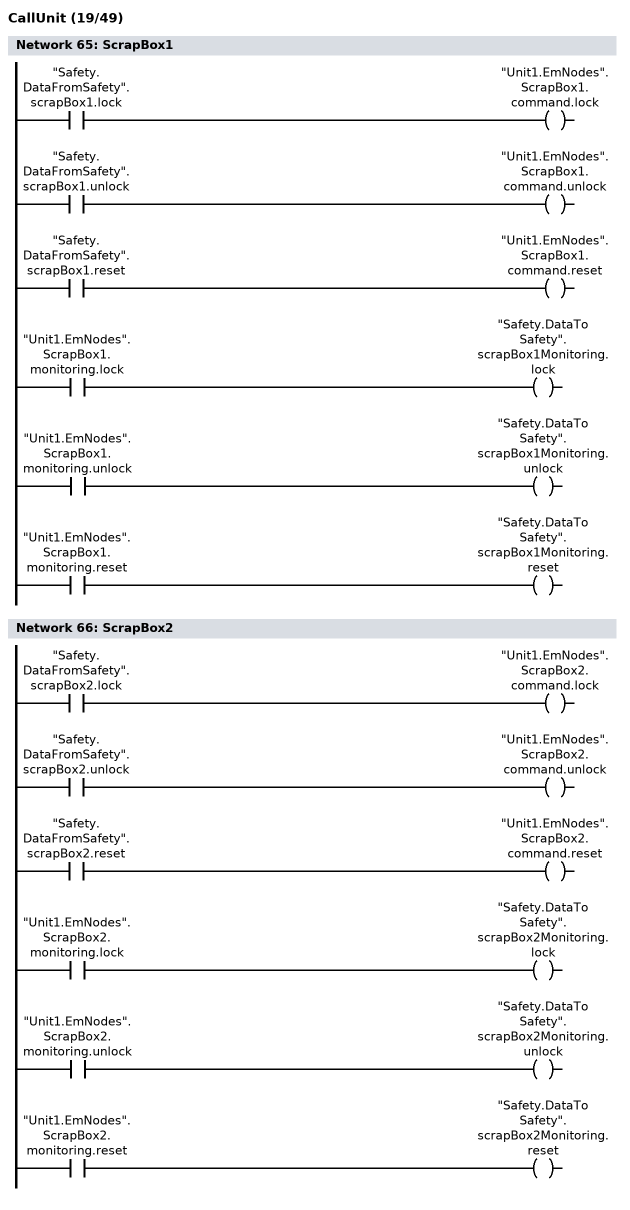
   RUNG wire#powerrail
      Contact( "Safety.DataFromSafety".scrapBox1.lock )
      Coil( "Unit1.EmNodes".ScrapBox1.command.lock )
   END_RUNG
   RUNG wire#powerrail
      Contact( "Safety.DataFromSafety".scrapBox1.unlock )
      Coil( "Unit1.EmNodes".ScrapBox1.command.unlock )
   END_RUNG
   RUNG wire#powerrail
      Contact( "Safety.DataFromSafety".scrapBox1.reset )
      Coil( "Unit1.EmNodes".ScrapBox1.command.reset )
   END_RUNG
   RUNG wire#powerrail
      Contact( "Unit1.EmNodes".ScrapBox1.monitoring.lock )
      Coil( "Safety.DataToSafety".scrapBox1Monitoring.lock )
   END_RUNG
   RUNG wire#powerrail
      Contact( "Unit1.EmNodes".ScrapBox1.monitoring.unlock )
      Coil( "Safety.DataToSafety".scrapBox1Monitoring.unlock )
   END_RUNG
   RUNG wire#powerrail
      Contact( "Unit1.EmNodes".ScrapBox1.monitoring.reset )
      Coil( "Safety.DataToSafety".scrapBox1Monitoring.reset )
   END_RUNG
   // the same network as SCL:
   "Unit1.EmNodes".ScrapBox1.command.lock := "Safety.DataFromSafety".scrapBox1.lock;
   "Unit1.EmNodes".ScrapBox1.command.unlock := "Safety.DataFromSafety".scrapBox1.unlock;
   "Unit1.EmNodes".ScrapBox1.command.reset := "Safety.DataFromSafety".scrapBox1.reset;
   "Safety.DataToSafety".scrapBox1Monitoring.lock := "Unit1.EmNodes".ScrapBox1.monitoring.lock;
   "Safety.DataToSafety".scrapBox1Monitoring.unlock := "Unit1.EmNodes".ScrapBox1.monitoring.unlock;
   "Safety.DataToSafety".scrapBox1Monitoring.reset := "Unit1.EmNodes".ScrapBox1.monitoring.reset;
END_REGION

REGION Network 66: ScrapBox2
   RUNG wire#powerrail
      Contact( "Safety.DataFromSafety".scrapBox2.lock )
      Coil( "Unit1.EmNodes".ScrapBox2.command.lock )
   END_RUNG
   RUNG wire#powerrail
      Contact( "Safety.DataFromSafety".scrapBox2.unlock )
      Coil( "Unit1.EmNodes".ScrapBox2.command.unlock )
   END_RUNG
   RUNG wire#powerrail
      Contact( "Safety.DataFromSafety".scrapBox2.reset )
      Coil( "Unit1.EmNodes".ScrapBox2.command.reset )
   END_RUNG
   RUNG wire#powerrail
      Contact( "Unit1.EmNodes".ScrapBox2.monitoring.lock )
      Coil( "Safety.DataToSafety".scrapBox2Monitoring.lock )
   END_RUNG
   RUNG wire#powerrail
      Contact( "Unit1.EmNodes".ScrapBox2.monitoring.unlock )
      Coil( "Safety.DataToSafety".scrapBox2Monitoring.unlock )
   END_RUNG
   RUNG wire#powerrail
      Contact( "Unit1.EmNodes".ScrapBox2.monitoring.reset )
      Coil( "Safety.DataToSafety".scrapBox2Monitoring.reset )
   END_RUNG
   // the same network as SCL:
   "Unit1.EmNodes".ScrapBox2.command.lock := "Safety.DataFromSafety".scrapBox2.lock;
   "Unit1.EmNodes".ScrapBox2.command.unlock := "Safety.DataFromSafety".scrapBox2.unlock;
   "Unit1.EmNodes".ScrapBox2.command.reset := "Safety.DataFromSafety".scrapBox2.reset;
   "Safety.DataToSafety".scrapBox2Monitoring.lock := "Unit1.EmNodes".ScrapBox2.monitoring.lock;
   "Safety.DataToSafety".scrapBox2Monitoring.unlock := "Unit1.EmNodes".ScrapBox2.monitoring.unlock;
   "Safety.DataToSafety".scrapBox2Monitoring.reset := "Unit1.EmNodes".ScrapBox2.monitoring.reset;
END_REGION

REGION Network 67: ScrapBox3
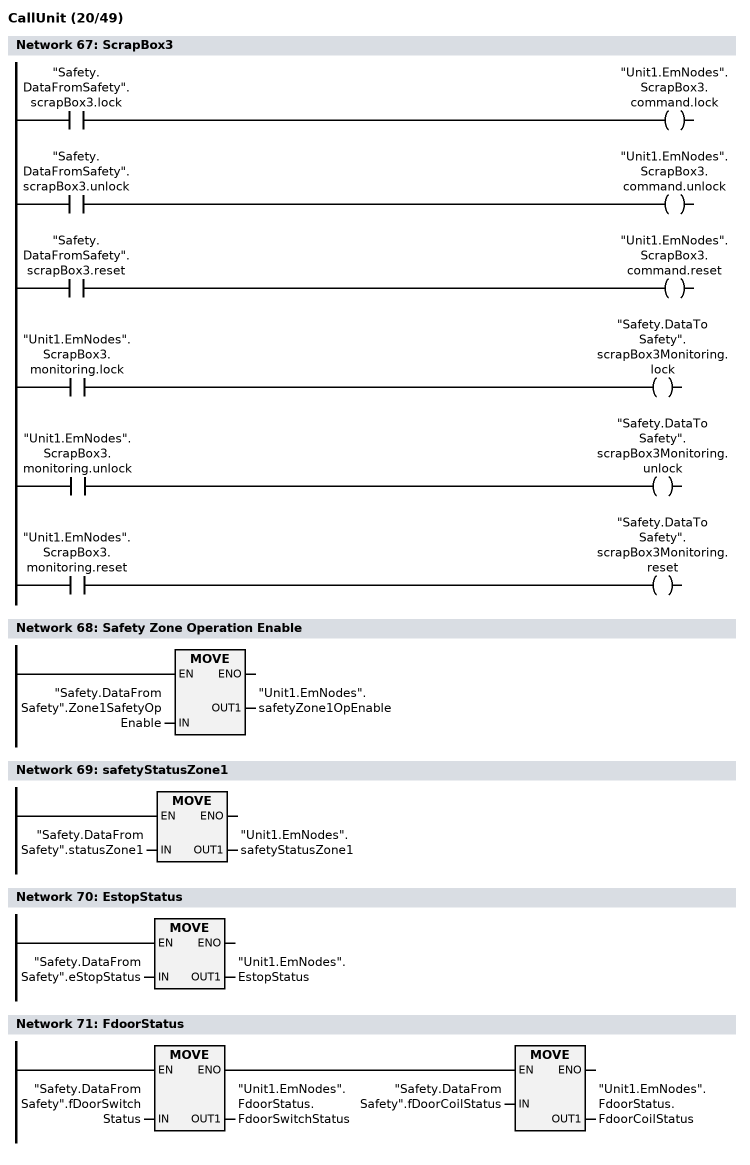
   RUNG wire#powerrail
      Contact( "Safety.DataFromSafety".scrapBox3.lock )
      Coil( "Unit1.EmNodes".ScrapBox3.command.lock )
   END_RUNG
   RUNG wire#powerrail
      Contact( "Safety.DataFromSafety".scrapBox3.unlock )
      Coil( "Unit1.EmNodes".ScrapBox3.command.unlock )
   END_RUNG
   RUNG wire#powerrail
      Contact( "Safety.DataFromSafety".scrapBox3.reset )
      Coil( "Unit1.EmNodes".ScrapBox3.command.reset )
   END_RUNG
   RUNG wire#powerrail
      Contact( "Unit1.EmNodes".ScrapBox3.monitoring.lock )
      Coil( "Safety.DataToSafety".scrapBox3Monitoring.lock )
   END_RUNG
   RUNG wire#powerrail
      Contact( "Unit1.EmNodes".ScrapBox3.monitoring.unlock )
      Coil( "Safety.DataToSafety".scrapBox3Monitoring.unlock )
   END_RUNG
   RUNG wire#powerrail
      Contact( "Unit1.EmNodes".ScrapBox3.monitoring.reset )
      Coil( "Safety.DataToSafety".scrapBox3Monitoring.reset )
   END_RUNG
   // the same network as SCL:
   "Unit1.EmNodes".ScrapBox3.command.lock := "Safety.DataFromSafety".scrapBox3.lock;
   "Unit1.EmNodes".ScrapBox3.command.unlock := "Safety.DataFromSafety".scrapBox3.unlock;
   "Unit1.EmNodes".ScrapBox3.command.reset := "Safety.DataFromSafety".scrapBox3.reset;
   "Safety.DataToSafety".scrapBox3Monitoring.lock := "Unit1.EmNodes".ScrapBox3.monitoring.lock;
   "Safety.DataToSafety".scrapBox3Monitoring.unlock := "Unit1.EmNodes".ScrapBox3.monitoring.unlock;
   "Safety.DataToSafety".scrapBox3Monitoring.reset := "Unit1.EmNodes".ScrapBox3.monitoring.reset;
END_REGION

REGION Network 68: Safety Zone Operation Enable
   RUNG wire#powerrail
      Move(in := "Safety.DataFromSafety".Zone1SafetyOpEnable, out1 => "Unit1.EmNodes".safetyZone1OpEnable)
   END_RUNG
   // the same network as SCL:
   "Unit1.EmNodes".safetyZone1OpEnable := "Safety.DataFromSafety".Zone1SafetyOpEnable;
END_REGION

REGION Network 69: safetyStatusZone1
   RUNG wire#powerrail
      Move(in := "Safety.DataFromSafety".statusZone1, out1 => "Unit1.EmNodes".safetyStatusZone1)
   END_RUNG
   // the same network as SCL:
   "Unit1.EmNodes".safetyStatusZone1 := "Safety.DataFromSafety".statusZone1;
END_REGION

REGION Network 70: EstopStatus
   RUNG wire#powerrail
      Move(in := "Safety.DataFromSafety".eStopStatus, out1 => "Unit1.EmNodes".EstopStatus)
   END_RUNG
   // the same network as SCL:
   "Unit1.EmNodes".EstopStatus := "Safety.DataFromSafety".eStopStatus;
END_REGION

REGION Network 71: FdoorStatus
   RUNG wire#powerrail
      Move(in := "Safety.DataFromSafety".fDoorSwitchStatus, out1 => "Unit1.EmNodes".FdoorStatus.FdoorSwitchStatus)
      Move(in := "Safety.DataFromSafety".fDoorCoilStatus, out1 => "Unit1.EmNodes".FdoorStatus.FdoorCoilStatus)
   END_RUNG
   // the same network as SCL:
   "Unit1.EmNodes".FdoorStatus.FdoorSwitchStatus := "Safety.DataFromSafety".fDoorSwitchStatus;
   "Unit1.EmNodes".FdoorStatus.FdoorCoilStatus := "Safety.DataFromSafety".fDoorCoilStatus;
END_REGION

REGION Network 72: Drive motion off
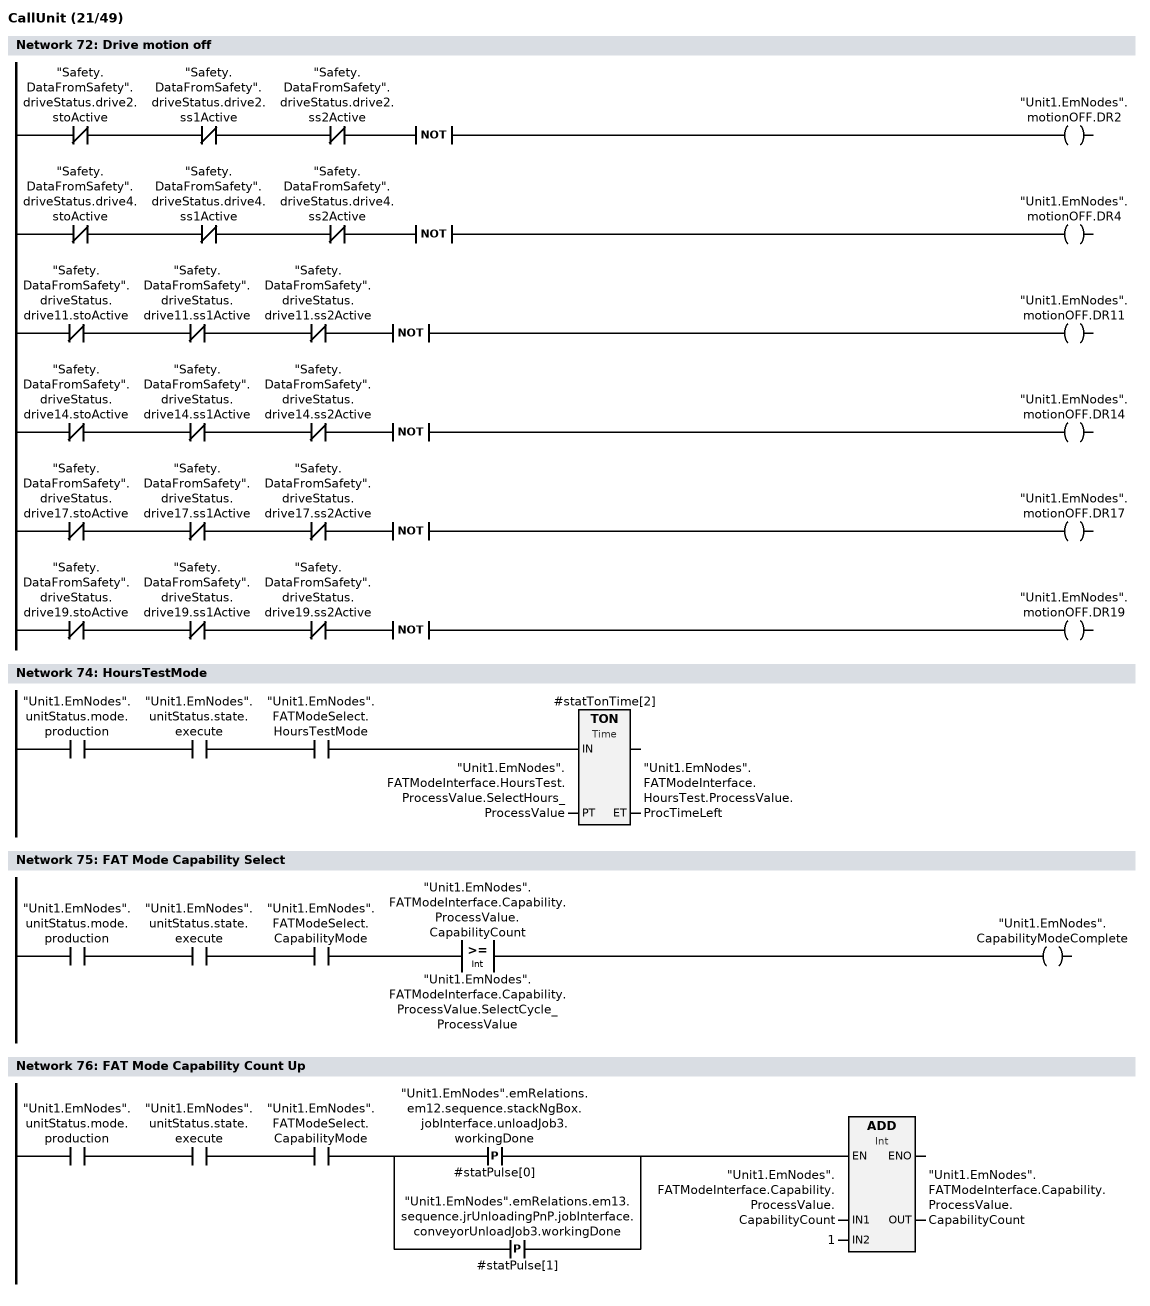
   RUNG wire#powerrail
      I_Contact( "Safety.DataFromSafety".driveStatus.drive2.stoActive )
      I_Contact( "Safety.DataFromSafety".driveStatus.drive2.ss1Active )
      I_Contact( "Safety.DataFromSafety".driveStatus.drive2.ss2Active )
      Not()
      Coil( "Unit1.EmNodes".motionOFF.DR2 )
   END_RUNG
   RUNG wire#powerrail
      I_Contact( "Safety.DataFromSafety".driveStatus.drive4.stoActive )
      I_Contact( "Safety.DataFromSafety".driveStatus.drive4.ss1Active )
      I_Contact( "Safety.DataFromSafety".driveStatus.drive4.ss2Active )
      Not()
      Coil( "Unit1.EmNodes".motionOFF.DR4 )
   END_RUNG
   RUNG wire#powerrail
      I_Contact( "Safety.DataFromSafety".driveStatus.drive11.stoActive )
      I_Contact( "Safety.DataFromSafety".driveStatus.drive11.ss1Active )
      I_Contact( "Safety.DataFromSafety".driveStatus.drive11.ss2Active )
      Not()
      Coil( "Unit1.EmNodes".motionOFF.DR11 )
   END_RUNG
   RUNG wire#powerrail
      I_Contact( "Safety.DataFromSafety".driveStatus.drive14.stoActive )
      I_Contact( "Safety.DataFromSafety".driveStatus.drive14.ss1Active )
      I_Contact( "Safety.DataFromSafety".driveStatus.drive14.ss2Active )
      Not()
      Coil( "Unit1.EmNodes".motionOFF.DR14 )
   END_RUNG
   RUNG wire#powerrail
      I_Contact( "Safety.DataFromSafety".driveStatus.drive17.stoActive )
      I_Contact( "Safety.DataFromSafety".driveStatus.drive17.ss1Active )
      I_Contact( "Safety.DataFromSafety".driveStatus.drive17.ss2Active )
      Not()
      Coil( "Unit1.EmNodes".motionOFF.DR17 )
   END_RUNG
   RUNG wire#powerrail
      I_Contact( "Safety.DataFromSafety".driveStatus.drive19.stoActive )
      I_Contact( "Safety.DataFromSafety".driveStatus.drive19.ss1Active )
      I_Contact( "Safety.DataFromSafety".driveStatus.drive19.ss2Active )
      Not()
      Coil( "Unit1.EmNodes".motionOFF.DR19 )
   END_RUNG
   // the same network as SCL:
   "Unit1.EmNodes".motionOFF.DR2 := NOT (NOT "Safety.DataFromSafety".driveStatus.drive2.stoActive AND NOT "Safety.DataFromSafety".driveStatus.drive2.ss1Active AND NOT "Safety.DataFromSafety".driveStatus.drive2.ss2Active);
   "Unit1.EmNodes".motionOFF.DR4 := NOT (NOT "Safety.DataFromSafety".driveStatus.drive4.stoActive AND NOT "Safety.DataFromSafety".driveStatus.drive4.ss1Active AND NOT "Safety.DataFromSafety".driveStatus.drive4.ss2Active);
   "Unit1.EmNodes".motionOFF.DR11 := NOT (NOT "Safety.DataFromSafety".driveStatus.drive11.stoActive AND NOT "Safety.DataFromSafety".driveStatus.drive11.ss1Active AND NOT "Safety.DataFromSafety".driveStatus.drive11.ss2Active);
   "Unit1.EmNodes".motionOFF.DR14 := NOT (NOT "Safety.DataFromSafety".driveStatus.drive14.stoActive AND NOT "Safety.DataFromSafety".driveStatus.drive14.ss1Active AND NOT "Safety.DataFromSafety".driveStatus.drive14.ss2Active);
   "Unit1.EmNodes".motionOFF.DR17 := NOT (NOT "Safety.DataFromSafety".driveStatus.drive17.stoActive AND NOT "Safety.DataFromSafety".driveStatus.drive17.ss1Active AND NOT "Safety.DataFromSafety".driveStatus.drive17.ss2Active);
   "Unit1.EmNodes".motionOFF.DR19 := NOT (NOT "Safety.DataFromSafety".driveStatus.drive19.stoActive AND NOT "Safety.DataFromSafety".driveStatus.drive19.ss1Active AND NOT "Safety.DataFromSafety".driveStatus.drive19.ss2Active);
END_REGION

REGION Network 73: ******************** FAT Mode ********************
END_REGION

REGION Network 74: HoursTestMode
   RUNG wire#powerrail
      Contact( "Unit1.EmNodes".unitStatus.mode.production )
      Contact( "Unit1.EmNodes".unitStatus.state.execute )
      Contact( "Unit1.EmNodes".FATModeSelect.HoursTestMode )
      { S7_Templates := "time_type := Time" } #statTonTime[2].TON(pt := "Unit1.EmNodes".FATModeInterface.HoursTest.ProcessValue.SelectHours_ProcessValue, et => "Unit1.EmNodes".FATModeInterface.HoursTest.ProcessValue.ProcTimeLeft)
   END_RUNG
   // the same network as SCL:
   #statTonTime[2].TON(IN := "Unit1.EmNodes".unitStatus.mode.production AND "Unit1.EmNodes".unitStatus.state.execute AND "Unit1.EmNodes".FATModeSelect.HoursTestMode,
                       PT := "Unit1.EmNodes".FATModeInterface.HoursTest.ProcessValue.SelectHours_ProcessValue,
                       ET => "Unit1.EmNodes".FATModeInterface.HoursTest.ProcessValue.ProcTimeLeft);
END_REGION

REGION Network 75: FAT Mode Capability Select
   RUNG wire#powerrail
      Contact( "Unit1.EmNodes".unitStatus.mode.production )
      Contact( "Unit1.EmNodes".unitStatus.state.execute )
      Contact( "Unit1.EmNodes".FATModeSelect.CapabilityMode )
      { S7_Templates := "SrcType := Int" } GE_Contact(in1 := "Unit1.EmNodes".FATModeInterface.Capability.ProcessValue.CapabilityCount, in2 := "Unit1.EmNodes".FATModeInterface.Capability.ProcessValue.SelectCycle_ProcessValue)
      Coil( "Unit1.EmNodes".CapabilityModeComplete )
   END_RUNG
   // the same network as SCL:
   "Unit1.EmNodes".CapabilityModeComplete := "Unit1.EmNodes".unitStatus.mode.production AND "Unit1.EmNodes".unitStatus.state.execute AND "Unit1.EmNodes".FATModeSelect.CapabilityMode AND ("Unit1.EmNodes".FATModeInterface.Capability.ProcessValue.CapabilityCount >= "Unit1.EmNodes".FATModeInterface.Capability.ProcessValue.SelectCycle_ProcessValue);
END_REGION

REGION Network 76: FAT Mode Capability Count Up
   RUNG wire#powerrail
      Contact( "Unit1.EmNodes".unitStatus.mode.production )
      Contact( "Unit1.EmNodes".unitStatus.state.execute )
      Contact( "Unit1.EmNodes".FATModeSelect.CapabilityMode )
      wire#w1
      P_Contact(operand := "Unit1.EmNodes".emRelations.em12.sequence.stackNgBox.jobInterface.unloadJob3.workingDone, bit := #statPulse[0])
      wire#w2
      { S7_Templates := "SrcType := Int" } Add(in1 := "Unit1.EmNodes".FATModeInterface.Capability.ProcessValue.CapabilityCount, in2 := 1, out => "Unit1.EmNodes".FATModeInterface.Capability.ProcessValue.CapabilityCount)
   END_RUNG
   RUNG wire#w1
      P_Contact(operand := "Unit1.EmNodes".emRelations.em13.sequence.jrUnloadingPnP.jobInterface.conveyorUnloadJob3.workingDone, bit := #statPulse[1])
   END_RUNG wire#w2
   // the same network as SCL:
   #_w1 := "Unit1.EmNodes".unitStatus.mode.production AND "Unit1.EmNodes".unitStatus.state.execute AND "Unit1.EmNodes".FATModeSelect.CapabilityMode AND "Unit1.EmNodes".emRelations.em12.sequence.stackNgBox.jobInterface.unloadJob3.workingDone AND NOT #statPulse[0];   // rising edge of "Unit1.EmNodes".emRelations.em12.sequence.stackNgBox.jobInterface.unloadJob3.workingDone
   #statPulse[0] := "Unit1.EmNodes".emRelations.em12.sequence.stackNgBox.jobInterface.unloadJob3.workingDone;
   #_w2 := "Unit1.EmNodes".unitStatus.mode.production AND "Unit1.EmNodes".unitStatus.state.execute AND "Unit1.EmNodes".FATModeSelect.CapabilityMode AND "Unit1.EmNodes".emRelations.em13.sequence.jrUnloadingPnP.jobInterface.conveyorUnloadJob3.workingDone AND NOT #statPulse[1];   // rising edge of "Unit1.EmNodes".emRelations.em13.sequence.jrUnloadingPnP.jobInterface.conveyorUnloadJob3.workingDone
   #statPulse[1] := "Unit1.EmNodes".emRelations.em13.sequence.jrUnloadingPnP.jobInterface.conveyorUnloadJob3.workingDone;
   IF #_w1 OR #_w2 THEN
       "Unit1.EmNodes".FATModeInterface.Capability.ProcessValue.CapabilityCount := "Unit1.EmNodes".FATModeInterface.Capability.ProcessValue.CapabilityCount + 1;
   END_IF;
END_REGION

REGION Network 77: FAT Mode Capability Count Clear
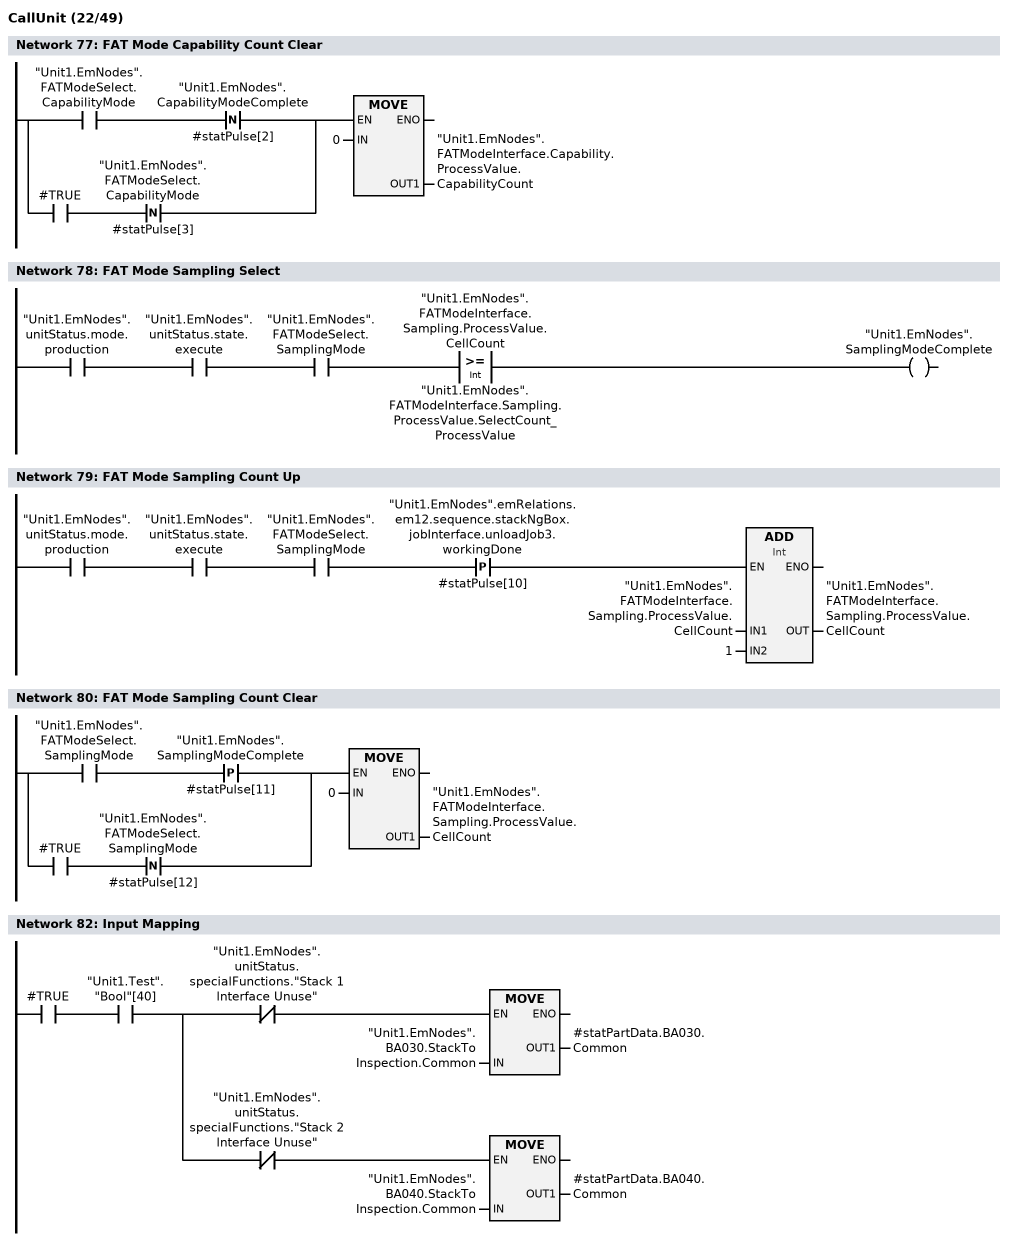
   RUNG wire#powerrail
      Contact( "Unit1.EmNodes".FATModeSelect.CapabilityMode )
      N_Contact(operand := "Unit1.EmNodes".CapabilityModeComplete, bit := #statPulse[2])
      wire#w1
      Move(in := 0, out1 => "Unit1.EmNodes".FATModeInterface.Capability.ProcessValue.CapabilityCount)
   END_RUNG
   RUNG wire#powerrail
      Contact( #TRUE )
      N_Contact(operand := "Unit1.EmNodes".FATModeSelect.CapabilityMode, bit := #statPulse[3])
   END_RUNG wire#w1
   // the same network as SCL:
   #_w1 := "Unit1.EmNodes".FATModeSelect.CapabilityMode AND NOT "Unit1.EmNodes".CapabilityModeComplete AND #statPulse[2];   // falling edge of "Unit1.EmNodes".CapabilityModeComplete
   #statPulse[2] := "Unit1.EmNodes".CapabilityModeComplete;
   #_w2 := #TRUE AND NOT "Unit1.EmNodes".FATModeSelect.CapabilityMode AND #statPulse[3];   // falling edge of "Unit1.EmNodes".FATModeSelect.CapabilityMode
   #statPulse[3] := "Unit1.EmNodes".FATModeSelect.CapabilityMode;
   IF #_w1 OR #_w2 THEN
       "Unit1.EmNodes".FATModeInterface.Capability.ProcessValue.CapabilityCount := 0;
   END_IF;
END_REGION

REGION Network 78: FAT Mode Sampling Select
   RUNG wire#powerrail
      Contact( "Unit1.EmNodes".unitStatus.mode.production )
      Contact( "Unit1.EmNodes".unitStatus.state.execute )
      Contact( "Unit1.EmNodes".FATModeSelect.SamplingMode )
      { S7_Templates := "SrcType := Int" } GE_Contact(in1 := "Unit1.EmNodes".FATModeInterface.Sampling.ProcessValue.CellCount, in2 := "Unit1.EmNodes".FATModeInterface.Sampling.ProcessValue.SelectCount_ProcessValue)
      Coil( "Unit1.EmNodes".SamplingModeComplete )
   END_RUNG
   // the same network as SCL:
   "Unit1.EmNodes".SamplingModeComplete := "Unit1.EmNodes".unitStatus.mode.production AND "Unit1.EmNodes".unitStatus.state.execute AND "Unit1.EmNodes".FATModeSelect.SamplingMode AND ("Unit1.EmNodes".FATModeInterface.Sampling.ProcessValue.CellCount >= "Unit1.EmNodes".FATModeInterface.Sampling.ProcessValue.SelectCount_ProcessValue);
END_REGION

REGION Network 79: FAT Mode Sampling Count Up
   RUNG wire#powerrail
      Contact( "Unit1.EmNodes".unitStatus.mode.production )
      Contact( "Unit1.EmNodes".unitStatus.state.execute )
      Contact( "Unit1.EmNodes".FATModeSelect.SamplingMode )
      P_Contact(operand := "Unit1.EmNodes".emRelations.em12.sequence.stackNgBox.jobInterface.unloadJob3.workingDone, bit := #statPulse[10])
      { S7_Templates := "SrcType := Int" } Add(in1 := "Unit1.EmNodes".FATModeInterface.Sampling.ProcessValue.CellCount, in2 := 1, out => "Unit1.EmNodes".FATModeInterface.Sampling.ProcessValue.CellCount)
   END_RUNG
   // the same network as SCL:
   #_w1 := "Unit1.EmNodes".unitStatus.mode.production AND "Unit1.EmNodes".unitStatus.state.execute AND "Unit1.EmNodes".FATModeSelect.SamplingMode AND "Unit1.EmNodes".emRelations.em12.sequence.stackNgBox.jobInterface.unloadJob3.workingDone AND NOT #statPulse[10];   // rising edge of "Unit1.EmNodes".emRelations.em12.sequence.stackNgBox.jobInterface.unloadJob3.workingDone
   #statPulse[10] := "Unit1.EmNodes".emRelations.em12.sequence.stackNgBox.jobInterface.unloadJob3.workingDone;
   IF #_w1 THEN
       "Unit1.EmNodes".FATModeInterface.Sampling.ProcessValue.CellCount := "Unit1.EmNodes".FATModeInterface.Sampling.ProcessValue.CellCount + 1;
   END_IF;
END_REGION

REGION Network 80: FAT Mode Sampling Count Clear
   RUNG wire#powerrail
      Contact( "Unit1.EmNodes".FATModeSelect.SamplingMode )
      P_Contact(operand := "Unit1.EmNodes".SamplingModeComplete, bit := #statPulse[11])
      wire#w1
      Move(in := 0, out1 => "Unit1.EmNodes".FATModeInterface.Sampling.ProcessValue.CellCount)
   END_RUNG
   RUNG wire#powerrail
      Contact( #TRUE )
      N_Contact(operand := "Unit1.EmNodes".FATModeSelect.SamplingMode, bit := #statPulse[12])
   END_RUNG wire#w1
   // the same network as SCL:
   #_w1 := "Unit1.EmNodes".FATModeSelect.SamplingMode AND "Unit1.EmNodes".SamplingModeComplete AND NOT #statPulse[11];   // rising edge of "Unit1.EmNodes".SamplingModeComplete
   #statPulse[11] := "Unit1.EmNodes".SamplingModeComplete;
   #_w2 := #TRUE AND NOT "Unit1.EmNodes".FATModeSelect.SamplingMode AND #statPulse[12];   // falling edge of "Unit1.EmNodes".FATModeSelect.SamplingMode
   #statPulse[12] := "Unit1.EmNodes".FATModeSelect.SamplingMode;
   IF #_w1 OR #_w2 THEN "Unit1.EmNodes".FATModeInterface.Sampling.ProcessValue.CellCount := 0; END_IF;
END_REGION

REGION Network 81: ******************** Part Data Mapping ********************
END_REGION

REGION Network 82: Input Mapping
   RUNG wire#powerrail
      Contact( #TRUE )
      Contact( "Unit1.Test"."Bool"[40] )
      wire#w1
      I_Contact( "Unit1.EmNodes".unitStatus.specialFunctions."Stack 1 lnterface Unuse" )
      Move(in := "Unit1.EmNodes".BA030.StackToInspection.Common, out1 => #statPartData.BA030.Common)
   END_RUNG
   RUNG wire#w1
      I_Contact( "Unit1.EmNodes".unitStatus.specialFunctions."Stack 2 lnterface Unuse" )
      Move(in := "Unit1.EmNodes".BA040.StackToInspection.Common, out1 => #statPartData.BA040.Common)
   END_RUNG
   // the same network as SCL:
   #_w1 := #TRUE AND "Unit1.Test"."Bool"[40];
   IF #_w1 AND NOT "Unit1.EmNodes".unitStatus.specialFunctions."Stack 1 lnterface Unuse" THEN
       #statPartData.BA030.Common := "Unit1.EmNodes".BA030.StackToInspection.Common;
   END_IF;
   IF #_w1 AND NOT "Unit1.EmNodes".unitStatus.specialFunctions."Stack 2 lnterface Unuse" THEN
       #statPartData.BA040.Common := "Unit1.EmNodes".BA040.StackToInspection.Common;
   END_IF;
END_REGION

REGION Network 83: Transfer P&P Left Job A/B Check
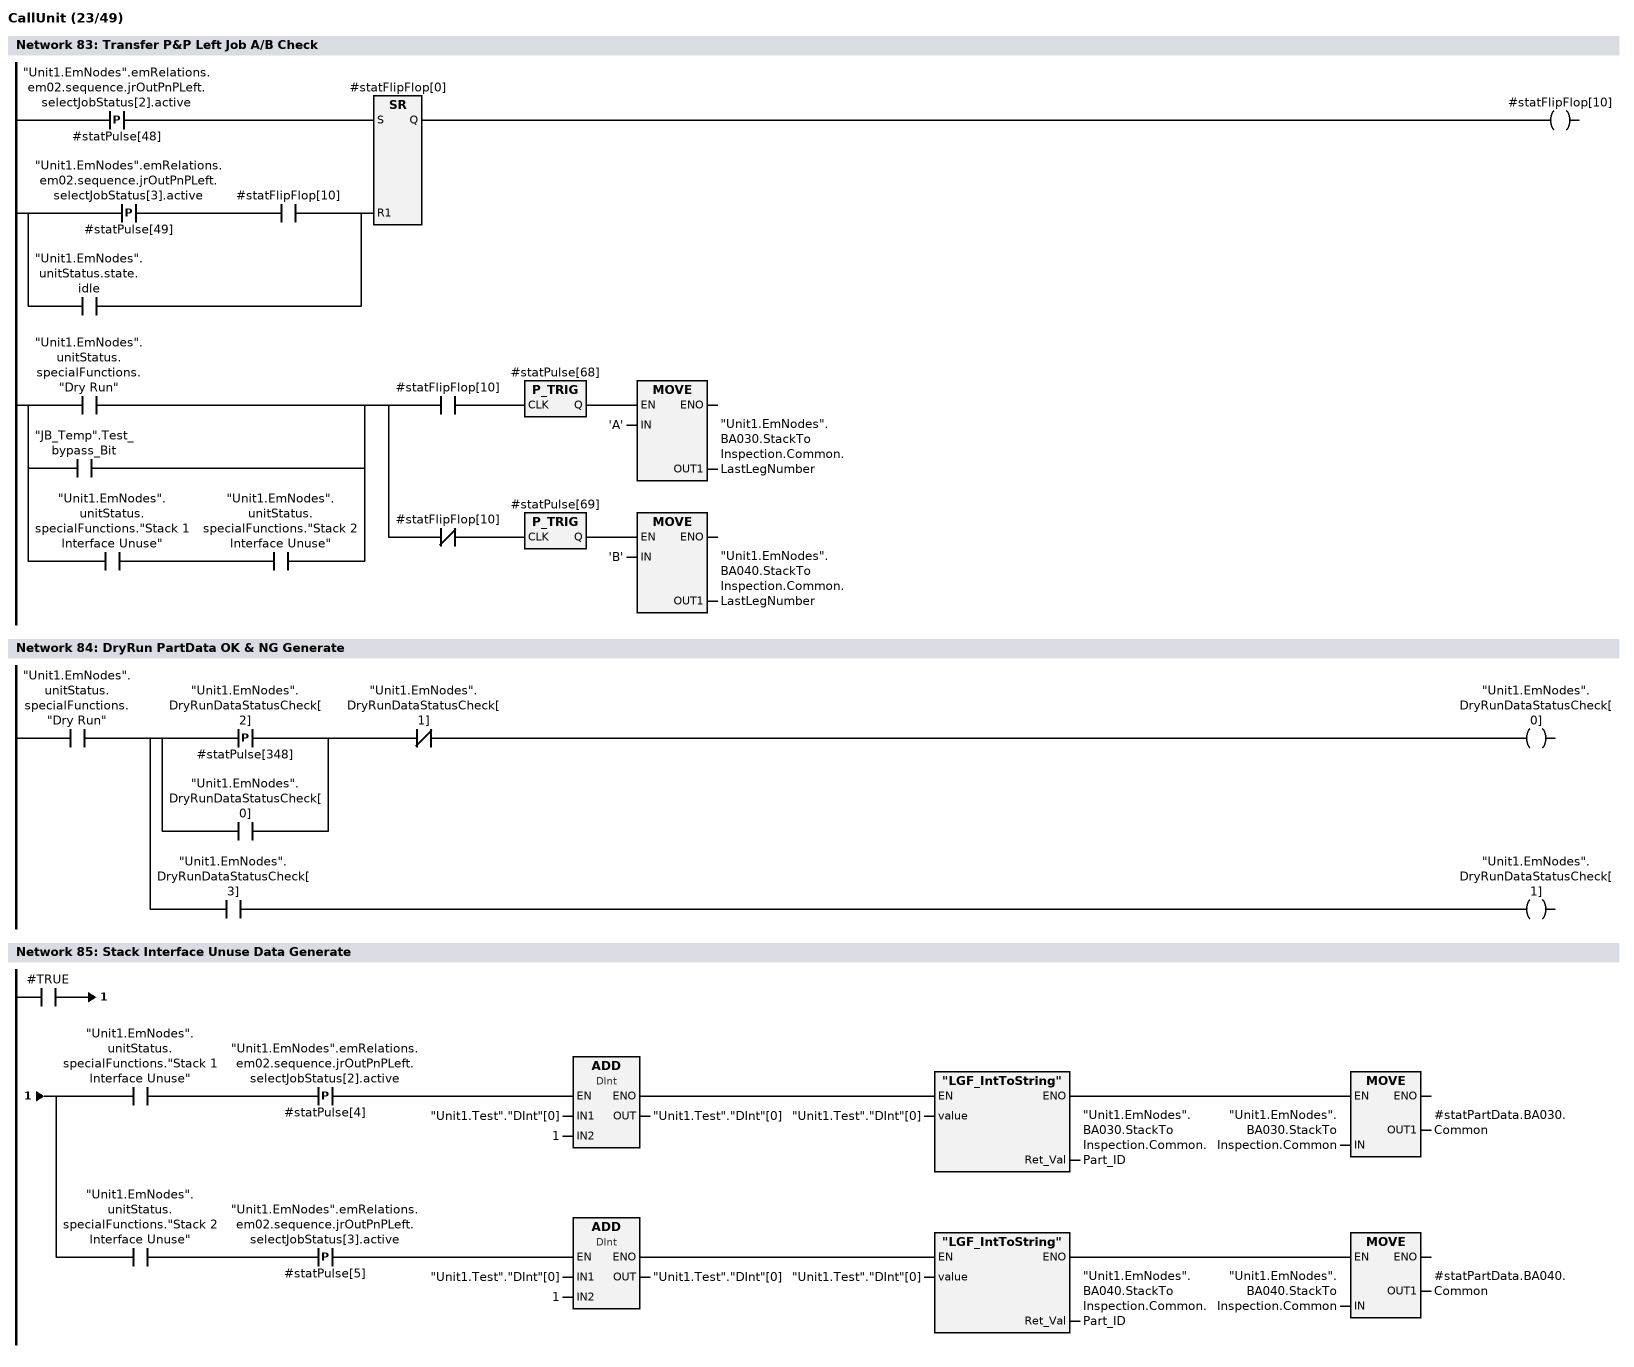
   RUNG wire#powerrail
      P_Contact(operand := "Unit1.EmNodes".emRelations.em02.sequence.jrOutPnPLeft.selectJobStatus[2].active, bit := #statPulse[48])
      S_SR(operand := #statFlipFlop[0], r1 := wire#w1)
      Coil( #statFlipFlop[10] )
   END_RUNG
   RUNG wire#powerrail
      P_Contact(operand := "Unit1.EmNodes".emRelations.em02.sequence.jrOutPnPLeft.selectJobStatus[3].active, bit := #statPulse[49])
      Contact( #statFlipFlop[10] )
   END_RUNG wire#w1
   RUNG wire#powerrail
      Contact( "Unit1.EmNodes".unitStatus.state.idle )
   END_RUNG wire#w1
   RUNG wire#powerrail
      Contact( "Unit1.EmNodes".unitStatus.specialFunctions."Dry Run" )
      wire#w2
      Contact( #statFlipFlop[10] )
      P_Trig( #statPulse[68] )
      Move(in := 'A', out1 => "Unit1.EmNodes".BA030.StackToInspection.Common.LastLegNumber)
   END_RUNG
   RUNG wire#powerrail
      Contact( "JB_Temp".Test_bypass_Bit )
   END_RUNG wire#w2
   RUNG wire#powerrail
      Contact( "Unit1.EmNodes".unitStatus.specialFunctions."Stack 1 lnterface Unuse" )
      Contact( "Unit1.EmNodes".unitStatus.specialFunctions."Stack 2 lnterface Unuse" )
   END_RUNG wire#w2
   RUNG wire#w2
      I_Contact( #statFlipFlop[10] )
      P_Trig( #statPulse[69] )
      Move(in := 'B', out1 => "Unit1.EmNodes".BA040.StackToInspection.Common.LastLegNumber)
   END_RUNG
   // the same network as SCL:
   #_w1 := "Unit1.EmNodes".emRelations.em02.sequence.jrOutPnPLeft.selectJobStatus[2].active AND NOT #statPulse[48];   // rising edge of "Unit1.EmNodes".emRelations.em02.sequence.jrOutPnPLeft.selectJobStatus[2].active
   #statPulse[48] := "Unit1.EmNodes".emRelations.em02.sequence.jrOutPnPLeft.selectJobStatus[2].active;
   #_w2 := "Unit1.EmNodes".emRelations.em02.sequence.jrOutPnPLeft.selectJobStatus[3].active AND NOT #statPulse[49];   // rising edge of "Unit1.EmNodes".emRelations.em02.sequence.jrOutPnPLeft.selectJobStatus[3].active
   #statPulse[49] := "Unit1.EmNodes".emRelations.em02.sequence.jrOutPnPLeft.selectJobStatus[3].active;
   #_w3 := (#_w2 AND #statFlipFlop[10]) OR "Unit1.EmNodes".unitStatus.state.idle;
   IF #_w1 THEN
       #statFlipFlop[0] := TRUE;   // SR flip-flop
   END_IF;
   IF #_w3 THEN #statFlipFlop[0] := FALSE; END_IF;
   #statFlipFlop[10] := #statFlipFlop[0];
   #_w4 := "Unit1.EmNodes".unitStatus.specialFunctions."Dry Run" OR "JB_Temp".Test_bypass_Bit OR ("Unit1.EmNodes".unitStatus.specialFunctions."Stack 1 lnterface Unuse" AND "Unit1.EmNodes".unitStatus.specialFunctions."Stack 2 lnterface Unuse");
   #_w5 := #_w4 AND #statFlipFlop[10];
   #_w6 := #_w5 AND NOT #statPulse[68];   // rising edge
   #statPulse[68] := #_w5;
   IF #_w6 THEN "Unit1.EmNodes".BA030.StackToInspection.Common.LastLegNumber := 'A'; END_IF;
   #_w7 := #_w4 AND NOT #statFlipFlop[10];
   #_w8 := #_w7 AND NOT #statPulse[69];   // rising edge
   #statPulse[69] := #_w7;
   IF #_w8 THEN "Unit1.EmNodes".BA040.StackToInspection.Common.LastLegNumber := 'B'; END_IF;
END_REGION

REGION Network 84: DryRun PartData OK & NG Generate
   RUNG wire#powerrail
      Contact( "Unit1.EmNodes".unitStatus.specialFunctions."Dry Run" )
      wire#w1
      P_Contact(operand := "Unit1.EmNodes".DryRunDataStatusCheck[2], bit := #statPulse[348])
      wire#w2
      I_Contact( "Unit1.EmNodes".DryRunDataStatusCheck[1] )
      Coil( "Unit1.EmNodes".DryRunDataStatusCheck[0] )
   END_RUNG
   RUNG wire#w1
      Contact( "Unit1.EmNodes".DryRunDataStatusCheck[0] )
   END_RUNG wire#w2
   RUNG wire#w1
      Contact( "Unit1.EmNodes".DryRunDataStatusCheck[3] )
      Coil( "Unit1.EmNodes".DryRunDataStatusCheck[1] )
   END_RUNG
   // the same network as SCL:
   #_w1 := "Unit1.EmNodes".unitStatus.specialFunctions."Dry Run" AND "Unit1.EmNodes".DryRunDataStatusCheck[2] AND NOT #statPulse[348];   // rising edge of "Unit1.EmNodes".DryRunDataStatusCheck[2]
   #statPulse[348] := "Unit1.EmNodes".DryRunDataStatusCheck[2];
   "Unit1.EmNodes".DryRunDataStatusCheck[0] := (#_w1 OR ("Unit1.EmNodes".unitStatus.specialFunctions."Dry Run" AND "Unit1.EmNodes".DryRunDataStatusCheck[0])) AND NOT "Unit1.EmNodes".DryRunDataStatusCheck[1];
   "Unit1.EmNodes".DryRunDataStatusCheck[1] := "Unit1.EmNodes".unitStatus.specialFunctions."Dry Run" AND "Unit1.EmNodes".DryRunDataStatusCheck[3];
END_REGION

REGION Network 85: Stack Interface Unuse Data Generate
   RUNG wire#powerrail
      Contact( #TRUE )
      wire#w1
      Contact( "Unit1.EmNodes".unitStatus.specialFunctions."Stack 1 lnterface Unuse" )
      P_Contact(operand := "Unit1.EmNodes".emRelations.em02.sequence.jrOutPnPLeft.selectJobStatus[2].active, bit := #statPulse[4])
      { S7_Templates := "SrcType := DInt" } Add(in1 := "Unit1.Test"."DInt"[0], in2 := 1, out => "Unit1.Test"."DInt"[0])
      "LGF_IntToString"(value := "Unit1.Test"."DInt"[0], Ret_Val => "Unit1.EmNodes".BA030.StackToInspection.Common.Part_ID)
      Move(in := "Unit1.EmNodes".BA030.StackToInspection.Common, out1 => #statPartData.BA030.Common)
   END_RUNG
   RUNG wire#w1
      Contact( "Unit1.EmNodes".unitStatus.specialFunctions."Stack 2 lnterface Unuse" )
      P_Contact(operand := "Unit1.EmNodes".emRelations.em02.sequence.jrOutPnPLeft.selectJobStatus[3].active, bit := #statPulse[5])
      { S7_Templates := "SrcType := DInt" } Add(in1 := "Unit1.Test"."DInt"[0], in2 := 1, out => "Unit1.Test"."DInt"[0])
      "LGF_IntToString"(value := "Unit1.Test"."DInt"[0], Ret_Val => "Unit1.EmNodes".BA040.StackToInspection.Common.Part_ID)
      Move(in := "Unit1.EmNodes".BA040.StackToInspection.Common, out1 => #statPartData.BA040.Common)
   END_RUNG
   // the same network as SCL:
   #_w1 := #TRUE AND "Unit1.EmNodes".unitStatus.specialFunctions."Stack 1 lnterface Unuse" AND "Unit1.EmNodes".emRelations.em02.sequence.jrOutPnPLeft.selectJobStatus[2].active AND NOT #statPulse[4];   // rising edge of "Unit1.EmNodes".emRelations.em02.sequence.jrOutPnPLeft.selectJobStatus[2].active
   #statPulse[4] := "Unit1.EmNodes".emRelations.em02.sequence.jrOutPnPLeft.selectJobStatus[2].active;
   IF #_w1 THEN "Unit1.Test"."DInt"[0] := "Unit1.Test"."DInt"[0] + 1; END_IF;
   "Unit1.EmNodes".BA030.StackToInspection.Common.Part_ID := "LGF_IntToString"(EN := #_w1,
                           value := "Unit1.Test"."DInt"[0],
                           ENO => #_w2);
   IF #_w2 THEN #statPartData.BA030.Common := "Unit1.EmNodes".BA030.StackToInspection.Common; END_IF;
   #_w3 := #TRUE AND "Unit1.EmNodes".unitStatus.specialFunctions."Stack 2 lnterface Unuse" AND "Unit1.EmNodes".emRelations.em02.sequence.jrOutPnPLeft.selectJobStatus[3].active AND NOT #statPulse[5];   // rising edge of "Unit1.EmNodes".emRelations.em02.sequence.jrOutPnPLeft.selectJobStatus[3].active
   #statPulse[5] := "Unit1.EmNodes".emRelations.em02.sequence.jrOutPnPLeft.selectJobStatus[3].active;
   IF #_w3 THEN "Unit1.Test"."DInt"[0] := "Unit1.Test"."DInt"[0] + 1; END_IF;
   "Unit1.EmNodes".BA040.StackToInspection.Common.Part_ID := "LGF_IntToString"(EN := #_w3,
                           value := "Unit1.Test"."DInt"[0],
                           ENO => #_w4);
   IF #_w4 THEN #statPartData.BA040.Common := "Unit1.EmNodes".BA040.StackToInspection.Common; END_IF;
END_REGION

REGION Network 86: Transfer And Generate Stack1 To JR Out P&P Left [BA030 → Em2]
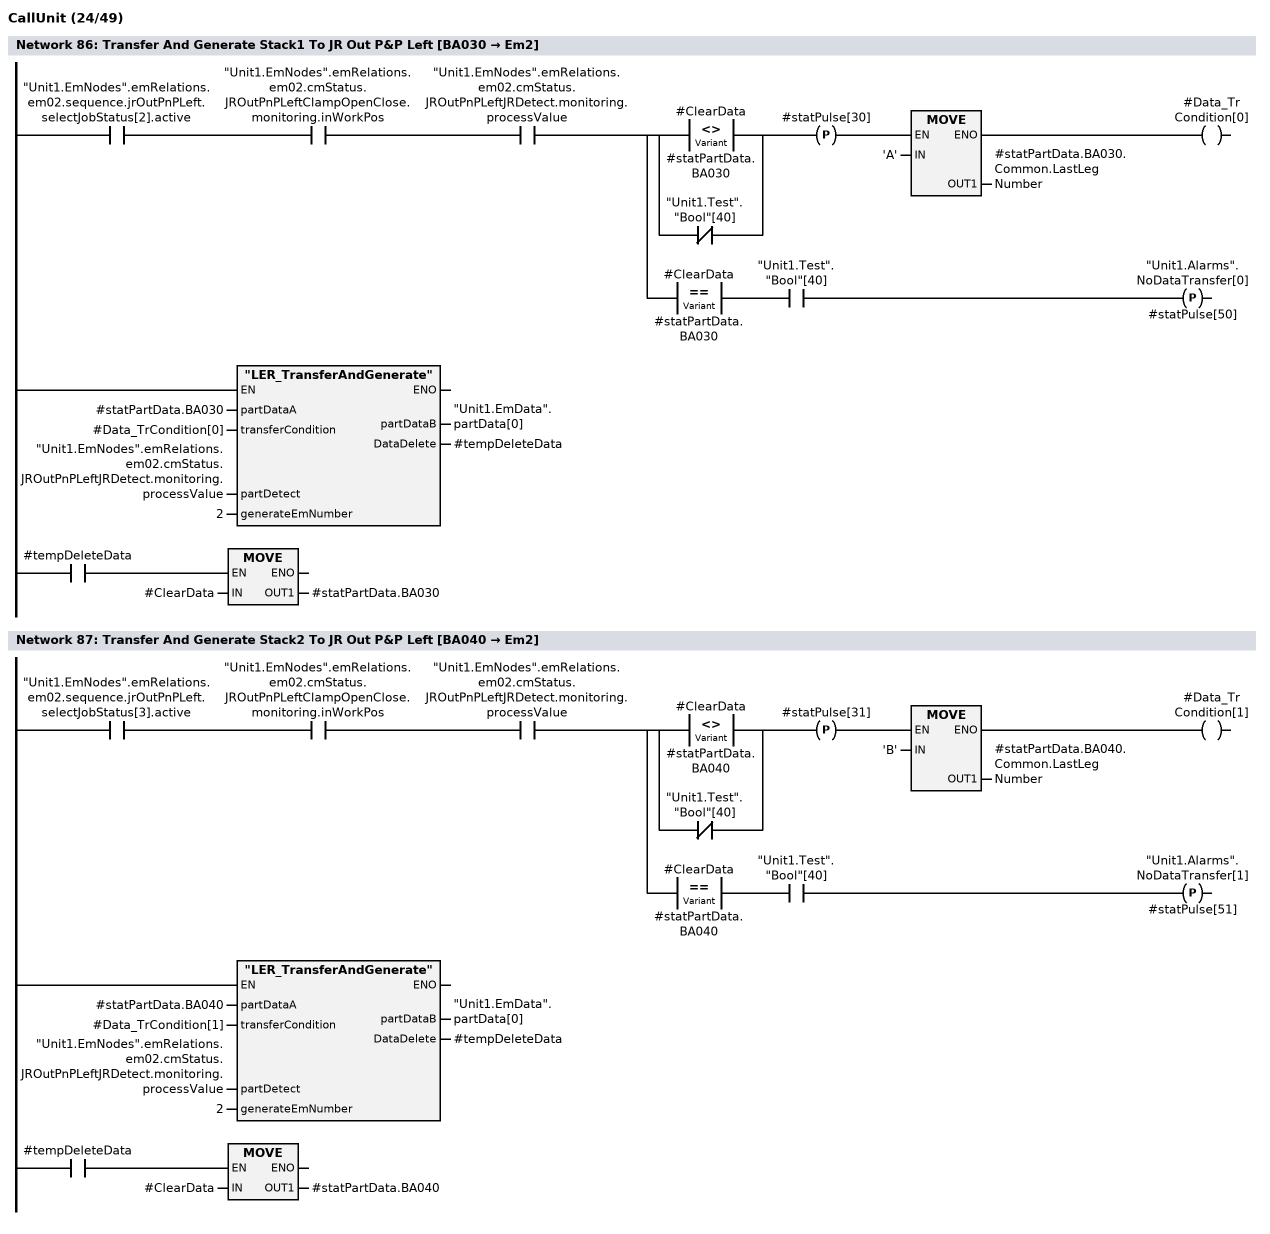
   #_w1 := "Unit1.EmNodes".emRelations.em02.sequence.jrOutPnPLeft.selectJobStatus[2].active AND "Unit1.EmNodes".emRelations.em02.cmStatus.JROutPnPLeftClampOpenClose.monitoring.inWorkPos AND "Unit1.EmNodes".emRelations.em02.cmStatus.JROutPnPLeftJRDetect.monitoring.processValue;
   #_w2 := #_w1 AND ((#ClearData <> #statPartData.BA030) OR NOT "Unit1.Test"."Bool"[40]);
   #_w3 := #_w2 AND NOT #statPulse[30];   // rising edge
   #statPulse[30] := #_w2;
   IF #_w3 THEN #statPartData.BA030.Common.LastLegNumber := 'A'; END_IF;
   #Data_TrCondition[0] := #_w3;
   #_w4 := #_w1 AND (#ClearData = #statPartData.BA030) AND "Unit1.Test"."Bool"[40];
   "Unit1.Alarms".NoDataTransfer[0] := #_w4 AND NOT #statPulse[50];   // rising edge
   #statPulse[50] := #_w4;
   "LER_TransferAndGenerate"(partDataA := #statPartData.BA030,
                           transferCondition := #Data_TrCondition[0],
                           partDetect := "Unit1.EmNodes".emRelations.em02.cmStatus.JROutPnPLeftJRDetect.monitoring.processValue,
                           generateEmNumber := 2,
                           partDataB => "Unit1.EmData".partData[0],
                           DataDelete => #tempDeleteData);
   IF #tempDeleteData THEN #statPartData.BA030 := #ClearData; END_IF;
END_REGION

REGION Network 87: Transfer And Generate Stack2 To JR Out P&P Left [BA040 → Em2]
   #_w1 := "Unit1.EmNodes".emRelations.em02.sequence.jrOutPnPLeft.selectJobStatus[3].active AND "Unit1.EmNodes".emRelations.em02.cmStatus.JROutPnPLeftClampOpenClose.monitoring.inWorkPos AND "Unit1.EmNodes".emRelations.em02.cmStatus.JROutPnPLeftJRDetect.monitoring.processValue;
   #_w2 := #_w1 AND ((#ClearData <> #statPartData.BA040) OR NOT "Unit1.Test"."Bool"[40]);
   #_w3 := #_w2 AND NOT #statPulse[31];   // rising edge
   #statPulse[31] := #_w2;
   IF #_w3 THEN #statPartData.BA040.Common.LastLegNumber := 'B'; END_IF;
   #Data_TrCondition[1] := #_w3;
   #_w4 := #_w1 AND (#ClearData = #statPartData.BA040) AND "Unit1.Test"."Bool"[40];
   "Unit1.Alarms".NoDataTransfer[1] := #_w4 AND NOT #statPulse[51];   // rising edge
   #statPulse[51] := #_w4;
   "LER_TransferAndGenerate"(partDataA := #statPartData.BA040,
                           transferCondition := #Data_TrCondition[1],
                           partDetect := "Unit1.EmNodes".emRelations.em02.cmStatus.JROutPnPLeftJRDetect.monitoring.processValue,
                           generateEmNumber := 2,
                           partDataB => "Unit1.EmData".partData[0],
                           DataDelete => #tempDeleteData);
   IF #tempDeleteData THEN #statPartData.BA040 := #ClearData; END_IF;
END_REGION

REGION Network 88: Transfer And Generate JR Out P&P Left To Top Tape [Em2 → Em3]
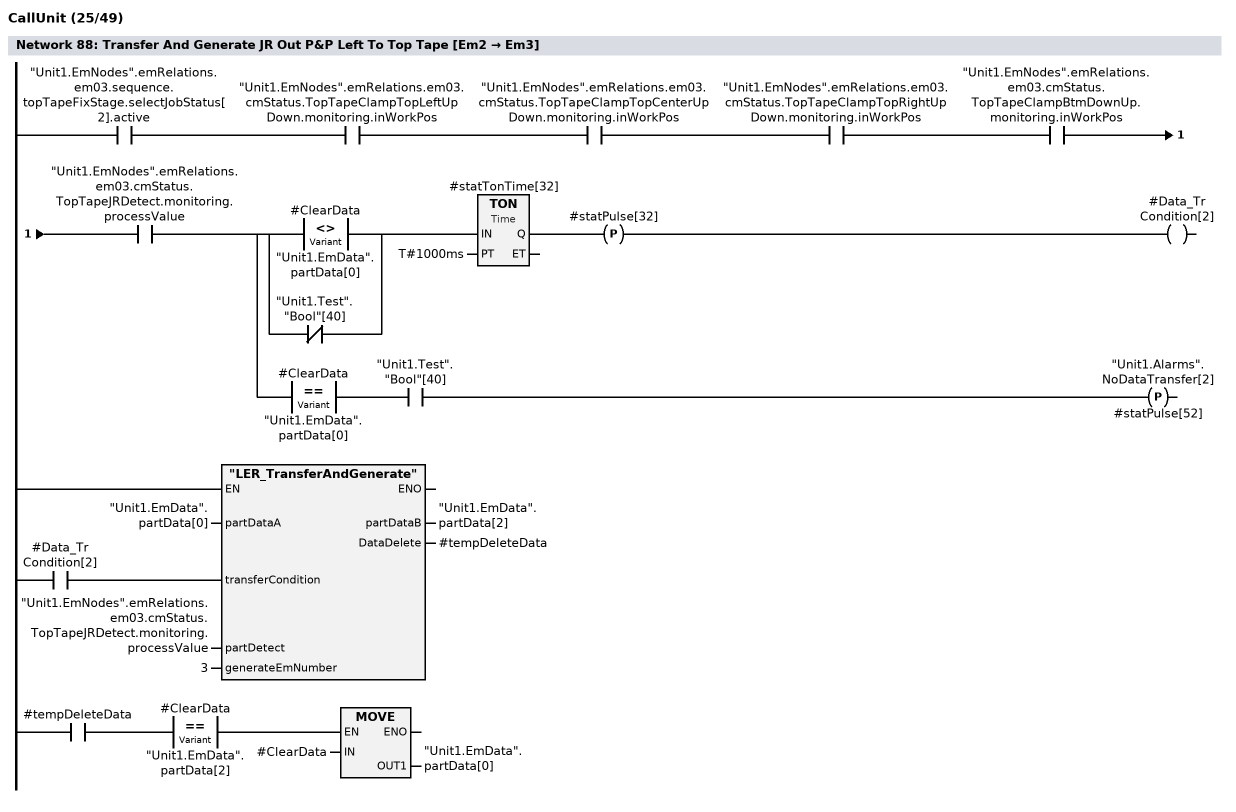
   #_w1 := "Unit1.EmNodes".emRelations.em03.sequence.topTapeFixStage.selectJobStatus[2].active AND "Unit1.EmNodes".emRelations.em03.cmStatus.TopTapeClampTopLeftUpDown.monitoring.inWorkPos AND "Unit1.EmNodes".emRelations.em03.cmStatus.TopTapeClampTopCenterUpDown.monitoring.inWorkPos AND "Unit1.EmNodes".emRelations.em03.cmStatus.TopTapeClampTopRightUpDown.monitoring.inWorkPos AND "Unit1.EmNodes".emRelations.em03.cmStatus.TopTapeClampBtmDownUp.monitoring.inWorkPos AND "Unit1.EmNodes".emRelations.em03.cmStatus.TopTapeJRDetect.monitoring.processValue;
   #statTonTime[32].TON(IN := #_w1 AND ((#ClearData <> "Unit1.EmData".partData[0]) OR NOT "Unit1.Test"."Bool"[40]),
                        PT := T#1000ms);
   #_w2 := #statTonTime[32].Q AND NOT #statPulse[32];   // rising edge
   #statPulse[32] := #statTonTime[32].Q;
   #Data_TrCondition[2] := #_w2;
   #_w3 := #_w1 AND (#ClearData = "Unit1.EmData".partData[0]) AND "Unit1.Test"."Bool"[40];
   "Unit1.Alarms".NoDataTransfer[2] := #_w3 AND NOT #statPulse[52];   // rising edge
   #statPulse[52] := #_w3;
   "LER_TransferAndGenerate"(partDataA := "Unit1.EmData".partData[0],
                           transferCondition := #Data_TrCondition[2],
                           partDetect := "Unit1.EmNodes".emRelations.em03.cmStatus.TopTapeJRDetect.monitoring.processValue,
                           generateEmNumber := 3,
                           partDataB => "Unit1.EmData".partData[2],
                           DataDelete => #tempDeleteData);
   IF #tempDeleteData AND (#ClearData = "Unit1.EmData".partData[2]) THEN
       "Unit1.EmData".partData[0] := #ClearData;
   END_IF;
END_REGION

REGION Network 89: Transfer And Generate Top Tape To JR Out P&P Right [Em3 → Em2]
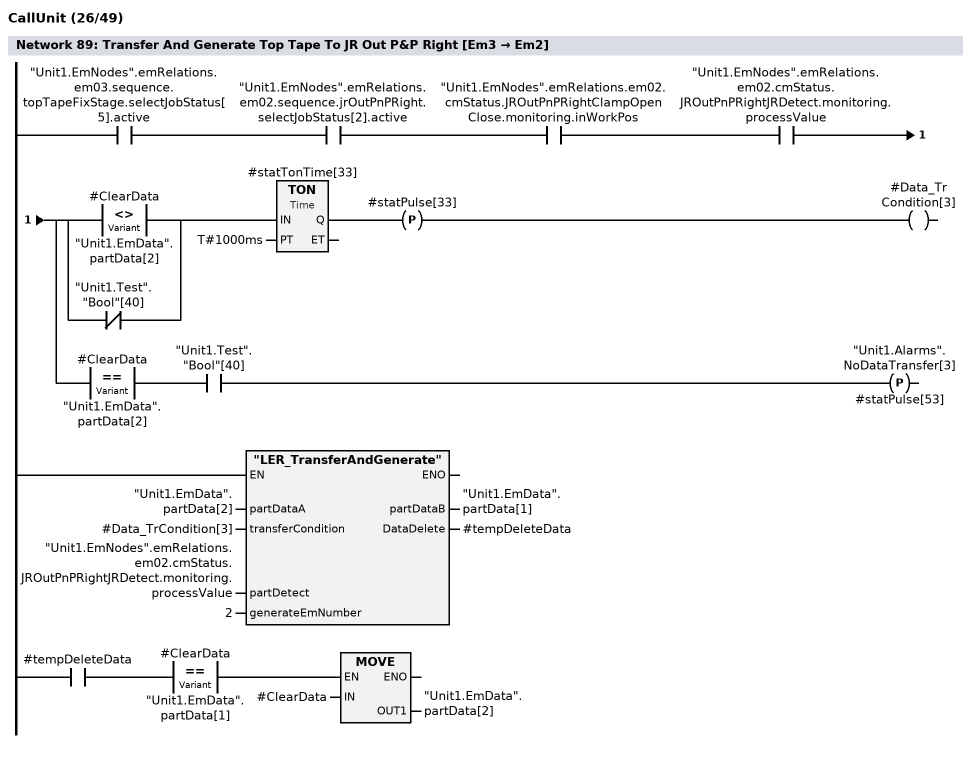
   #_w1 := "Unit1.EmNodes".emRelations.em03.sequence.topTapeFixStage.selectJobStatus[5].active AND "Unit1.EmNodes".emRelations.em02.sequence.jrOutPnPRight.selectJobStatus[2].active AND "Unit1.EmNodes".emRelations.em02.cmStatus.JROutPnPRightClampOpenClose.monitoring.inWorkPos AND "Unit1.EmNodes".emRelations.em02.cmStatus.JROutPnPRightJRDetect.monitoring.processValue;
   #statTonTime[33].TON(IN := #_w1 AND ((#ClearData <> "Unit1.EmData".partData[2]) OR NOT "Unit1.Test"."Bool"[40]),
                        PT := T#1000ms);
   #_w2 := #statTonTime[33].Q AND NOT #statPulse[33];   // rising edge
   #statPulse[33] := #statTonTime[33].Q;
   #Data_TrCondition[3] := #_w2;
   #_w3 := #_w1 AND (#ClearData = "Unit1.EmData".partData[2]) AND "Unit1.Test"."Bool"[40];
   "Unit1.Alarms".NoDataTransfer[3] := #_w3 AND NOT #statPulse[53];   // rising edge
   #statPulse[53] := #_w3;
   "LER_TransferAndGenerate"(partDataA := "Unit1.EmData".partData[2],
                           transferCondition := #Data_TrCondition[3],
                           partDetect := "Unit1.EmNodes".emRelations.em02.cmStatus.JROutPnPRightJRDetect.monitoring.processValue,
                           generateEmNumber := 2,
                           partDataB => "Unit1.EmData".partData[1],
                           DataDelete => #tempDeleteData);
   IF #tempDeleteData AND (#ClearData = "Unit1.EmData".partData[1]) THEN
       "Unit1.EmData".partData[2] := #ClearData;
   END_IF;
END_REGION

REGION Network 90: Transfer And Generate JR Out P&P Right To Side Tape [Em2 → Em4]
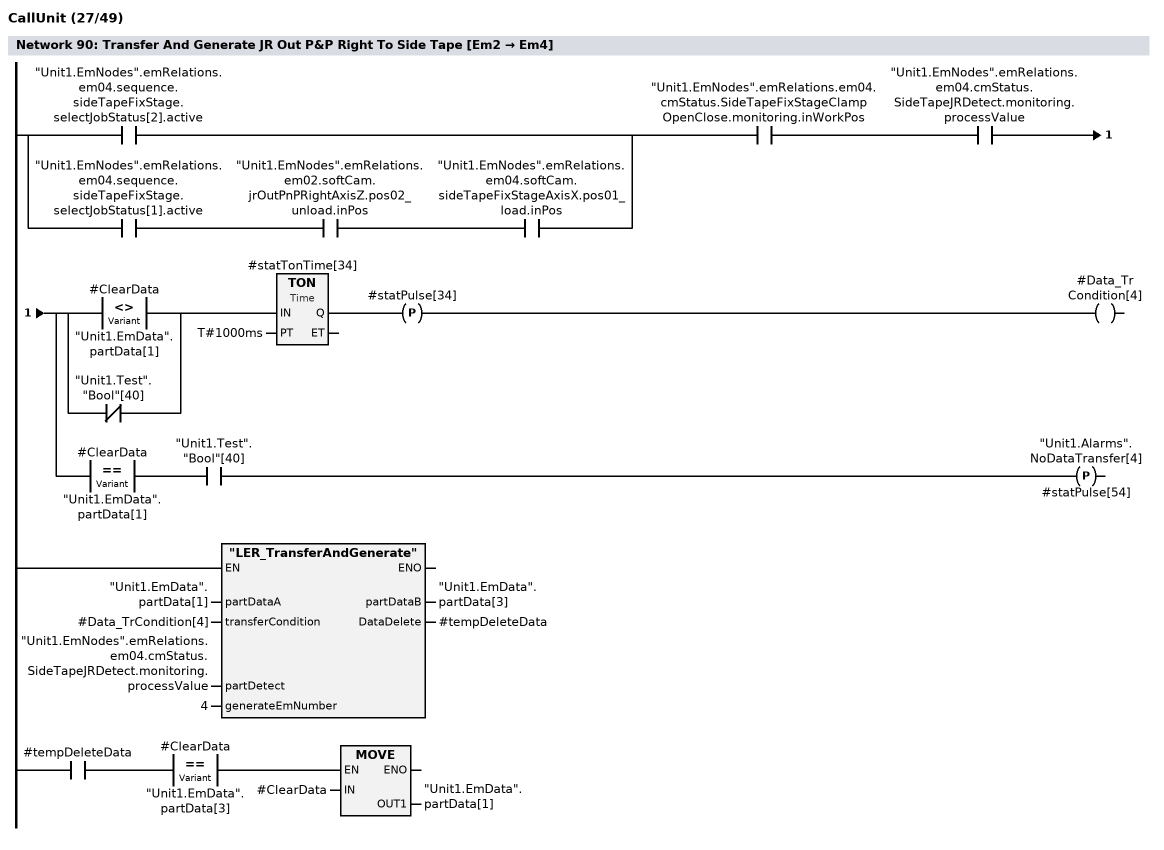
   #_w1 := ("Unit1.EmNodes".emRelations.em04.sequence.sideTapeFixStage.selectJobStatus[2].active OR ("Unit1.EmNodes".emRelations.em04.sequence.sideTapeFixStage.selectJobStatus[1].active AND "Unit1.EmNodes".emRelations.em02.softCam.jrOutPnPRightAxisZ.pos02_unload.inPos AND "Unit1.EmNodes".emRelations.em04.softCam.sideTapeFixStageAxisX.pos01_load.inPos)) AND "Unit1.EmNodes".emRelations.em04.cmStatus.SideTapeFixStageClampOpenClose.monitoring.inWorkPos AND "Unit1.EmNodes".emRelations.em04.cmStatus.SideTapeJRDetect.monitoring.processValue;
   #statTonTime[34].TON(IN := #_w1 AND ((#ClearData <> "Unit1.EmData".partData[1]) OR NOT "Unit1.Test"."Bool"[40]),
                        PT := T#1000ms);
   #_w2 := #statTonTime[34].Q AND NOT #statPulse[34];   // rising edge
   #statPulse[34] := #statTonTime[34].Q;
   #Data_TrCondition[4] := #_w2;
   #_w3 := #_w1 AND (#ClearData = "Unit1.EmData".partData[1]) AND "Unit1.Test"."Bool"[40];
   "Unit1.Alarms".NoDataTransfer[4] := #_w3 AND NOT #statPulse[54];   // rising edge
   #statPulse[54] := #_w3;
   "LER_TransferAndGenerate"(partDataA := "Unit1.EmData".partData[1],
                           transferCondition := #Data_TrCondition[4],
                           partDetect := "Unit1.EmNodes".emRelations.em04.cmStatus.SideTapeJRDetect.monitoring.processValue,
                           generateEmNumber := 4,
                           partDataB => "Unit1.EmData".partData[3],
                           DataDelete => #tempDeleteData);
   IF #tempDeleteData AND (#ClearData = "Unit1.EmData".partData[3]) THEN
       "Unit1.EmData".partData[1] := #ClearData;
   END_IF;
END_REGION

REGION Network 91: Transfer And Generate Side Tape To Transfer P&P Left [Em4 → Em5]
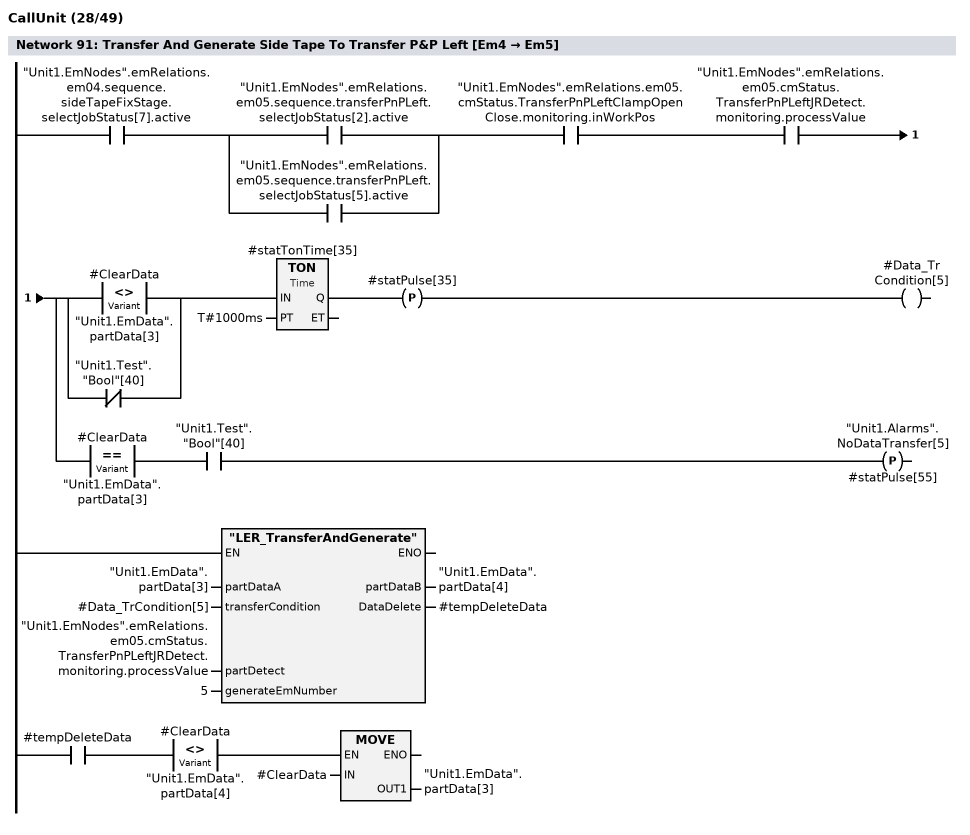
   #_w1 := "Unit1.EmNodes".emRelations.em04.sequence.sideTapeFixStage.selectJobStatus[7].active AND ("Unit1.EmNodes".emRelations.em05.sequence.transferPnPLeft.selectJobStatus[2].active OR "Unit1.EmNodes".emRelations.em05.sequence.transferPnPLeft.selectJobStatus[5].active) AND "Unit1.EmNodes".emRelations.em05.cmStatus.TransferPnPLeftClampOpenClose.monitoring.inWorkPos AND "Unit1.EmNodes".emRelations.em05.cmStatus.TransferPnPLeftJRDetect.monitoring.processValue;
   #statTonTime[35].TON(IN := #_w1 AND ((#ClearData <> "Unit1.EmData".partData[3]) OR NOT "Unit1.Test"."Bool"[40]),
                        PT := T#1000ms);
   #_w2 := #statTonTime[35].Q AND NOT #statPulse[35];   // rising edge
   #statPulse[35] := #statTonTime[35].Q;
   #Data_TrCondition[5] := #_w2;
   #_w3 := #_w1 AND (#ClearData = "Unit1.EmData".partData[3]) AND "Unit1.Test"."Bool"[40];
   "Unit1.Alarms".NoDataTransfer[5] := #_w3 AND NOT #statPulse[55];   // rising edge
   #statPulse[55] := #_w3;
   "LER_TransferAndGenerate"(partDataA := "Unit1.EmData".partData[3],
                           transferCondition := #Data_TrCondition[5],
                           partDetect := "Unit1.EmNodes".emRelations.em05.cmStatus.TransferPnPLeftJRDetect.monitoring.processValue,
                           generateEmNumber := 5,
                           partDataB => "Unit1.EmData".partData[4],
                           DataDelete => #tempDeleteData);
   IF #tempDeleteData AND (#ClearData <> "Unit1.EmData".partData[4]) THEN
       "Unit1.EmData".partData[3] := #ClearData;
   END_IF;
END_REGION

REGION Network 92: Transfer And Generate Transfer P&P Left To Hot Press Left [Em5 → Em6]
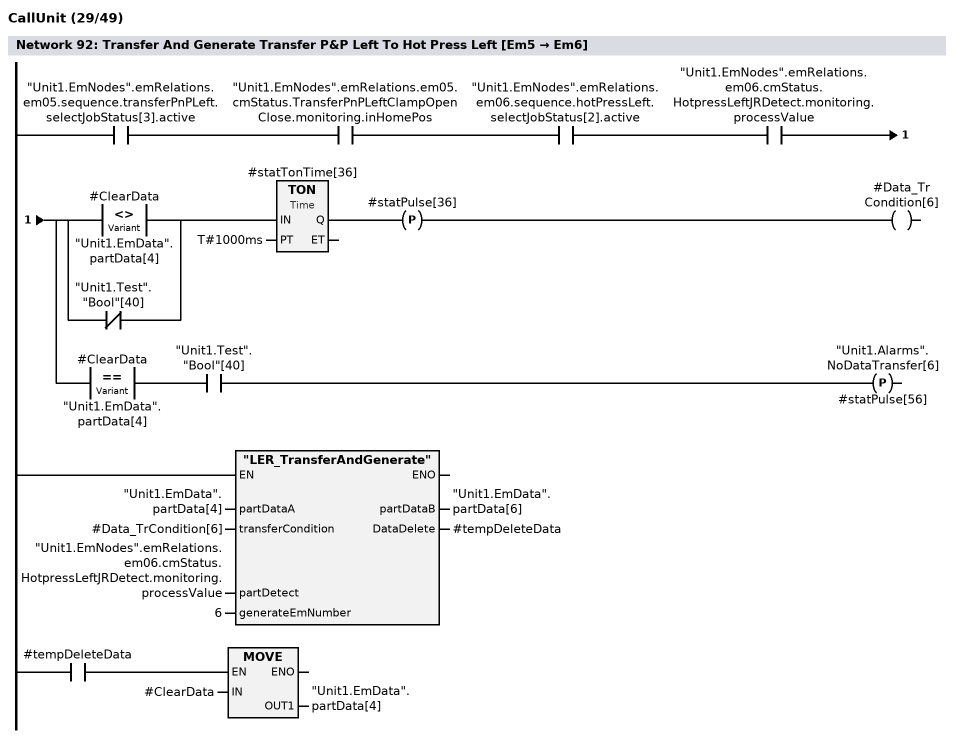
   #_w1 := "Unit1.EmNodes".emRelations.em05.sequence.transferPnPLeft.selectJobStatus[3].active AND "Unit1.EmNodes".emRelations.em05.cmStatus.TransferPnPLeftClampOpenClose.monitoring.inHomePos AND "Unit1.EmNodes".emRelations.em06.sequence.hotPressLeft.selectJobStatus[2].active AND "Unit1.EmNodes".emRelations.em06.cmStatus.HotpressLeftJRDetect.monitoring.processValue;
   #statTonTime[36].TON(IN := #_w1 AND ((#ClearData <> "Unit1.EmData".partData[4]) OR NOT "Unit1.Test"."Bool"[40]),
                        PT := T#1000ms);
   #_w2 := #statTonTime[36].Q AND NOT #statPulse[36];   // rising edge
   #statPulse[36] := #statTonTime[36].Q;
   #Data_TrCondition[6] := #_w2;
   #_w3 := #_w1 AND (#ClearData = "Unit1.EmData".partData[4]) AND "Unit1.Test"."Bool"[40];
   "Unit1.Alarms".NoDataTransfer[6] := #_w3 AND NOT #statPulse[56];   // rising edge
   #statPulse[56] := #_w3;
   "LER_TransferAndGenerate"(partDataA := "Unit1.EmData".partData[4],
                           transferCondition := #Data_TrCondition[6],
                           partDetect := "Unit1.EmNodes".emRelations.em06.cmStatus.HotpressLeftJRDetect.monitoring.processValue,
                           generateEmNumber := 6,
                           partDataB => "Unit1.EmData".partData[6],
                           DataDelete => #tempDeleteData);
   IF #tempDeleteData THEN "Unit1.EmData".partData[4] := #ClearData; END_IF;
END_REGION

REGION Network 93: Transfer And Generate Hot Press Left To Transfer P&P Left [Em6 → Em5]
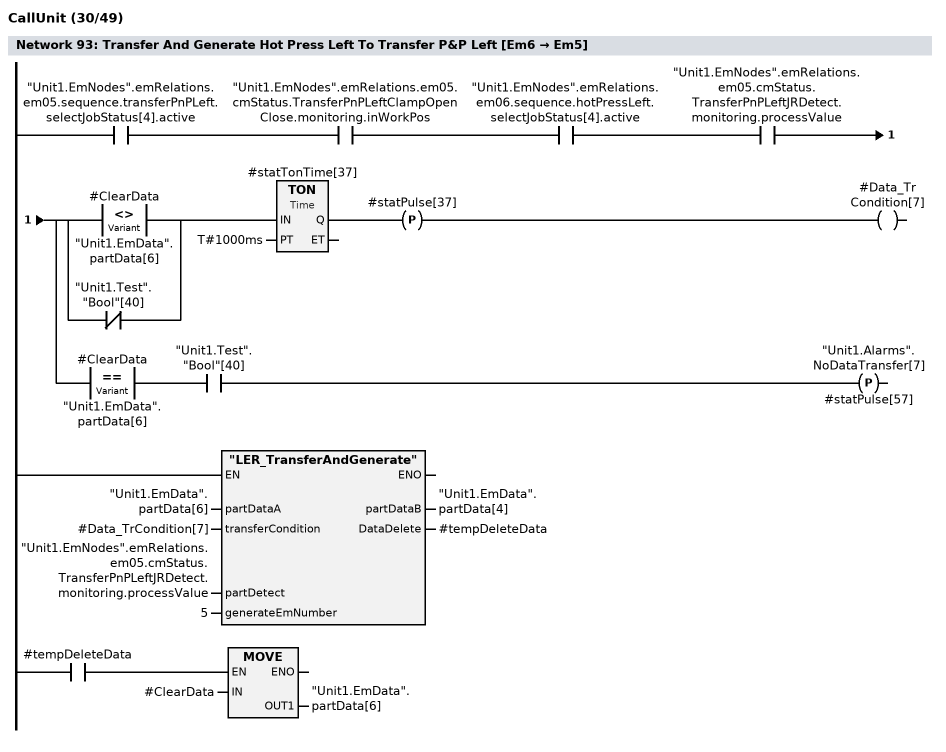
   #_w1 := "Unit1.EmNodes".emRelations.em05.sequence.transferPnPLeft.selectJobStatus[4].active AND "Unit1.EmNodes".emRelations.em05.cmStatus.TransferPnPLeftClampOpenClose.monitoring.inWorkPos AND "Unit1.EmNodes".emRelations.em06.sequence.hotPressLeft.selectJobStatus[4].active AND "Unit1.EmNodes".emRelations.em05.cmStatus.TransferPnPLeftJRDetect.monitoring.processValue;
   #statTonTime[37].TON(IN := #_w1 AND ((#ClearData <> "Unit1.EmData".partData[6]) OR NOT "Unit1.Test"."Bool"[40]),
                        PT := T#1000ms);
   #_w2 := #statTonTime[37].Q AND NOT #statPulse[37];   // rising edge
   #statPulse[37] := #statTonTime[37].Q;
   #Data_TrCondition[7] := #_w2;
   #_w3 := #_w1 AND (#ClearData = "Unit1.EmData".partData[6]) AND "Unit1.Test"."Bool"[40];
   "Unit1.Alarms".NoDataTransfer[7] := #_w3 AND NOT #statPulse[57];   // rising edge
   #statPulse[57] := #_w3;
   "LER_TransferAndGenerate"(partDataA := "Unit1.EmData".partData[6],
                           transferCondition := #Data_TrCondition[7],
                           partDetect := "Unit1.EmNodes".emRelations.em05.cmStatus.TransferPnPLeftJRDetect.monitoring.processValue,
                           generateEmNumber := 5,
                           partDataB => "Unit1.EmData".partData[4],
                           DataDelete => #tempDeleteData);
   IF #tempDeleteData THEN "Unit1.EmData".partData[6] := #ClearData; END_IF;
END_REGION

REGION Network 94: Transfer And Generate Transfer P&P Left To Hot Press Right [Em5 → Em7]
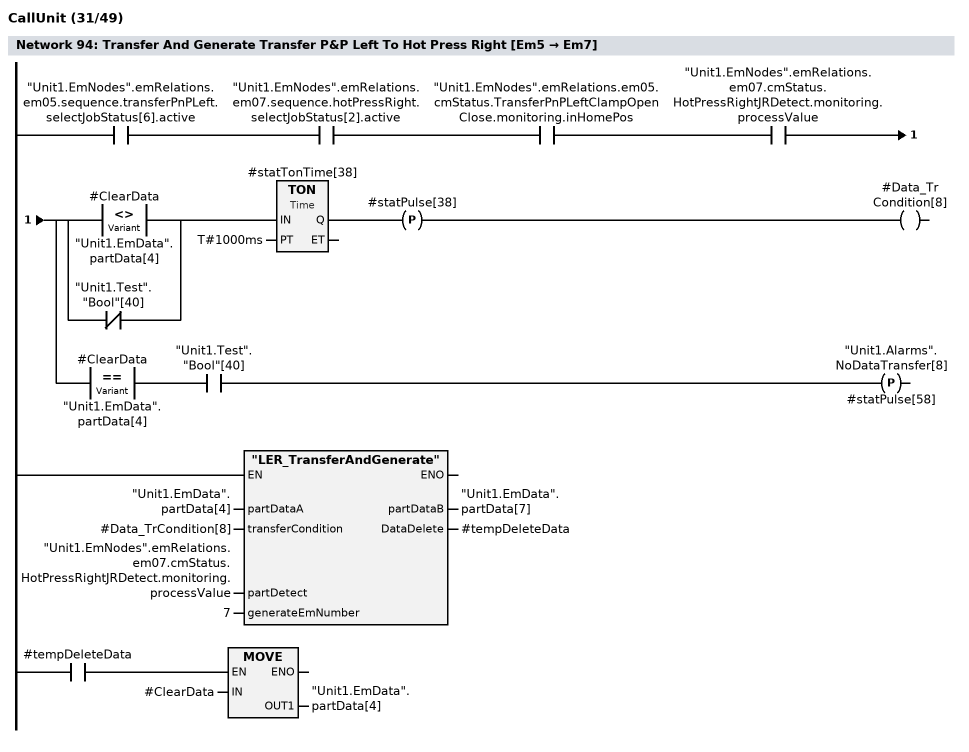
   #_w1 := "Unit1.EmNodes".emRelations.em05.sequence.transferPnPLeft.selectJobStatus[6].active AND "Unit1.EmNodes".emRelations.em07.sequence.hotPressRight.selectJobStatus[2].active AND "Unit1.EmNodes".emRelations.em05.cmStatus.TransferPnPLeftClampOpenClose.monitoring.inHomePos AND "Unit1.EmNodes".emRelations.em07.cmStatus.HotPressRightJRDetect.monitoring.processValue;
   #statTonTime[38].TON(IN := #_w1 AND ((#ClearData <> "Unit1.EmData".partData[4]) OR NOT "Unit1.Test"."Bool"[40]),
                        PT := T#1000ms);
   #_w2 := #statTonTime[38].Q AND NOT #statPulse[38];   // rising edge
   #statPulse[38] := #statTonTime[38].Q;
   #Data_TrCondition[8] := #_w2;
   #_w3 := #_w1 AND (#ClearData = "Unit1.EmData".partData[4]) AND "Unit1.Test"."Bool"[40];
   "Unit1.Alarms".NoDataTransfer[8] := #_w3 AND NOT #statPulse[58];   // rising edge
   #statPulse[58] := #_w3;
   "LER_TransferAndGenerate"(partDataA := "Unit1.EmData".partData[4],
                           transferCondition := #Data_TrCondition[8],
                           partDetect := "Unit1.EmNodes".emRelations.em07.cmStatus.HotPressRightJRDetect.monitoring.processValue,
                           generateEmNumber := 7,
                           partDataB => "Unit1.EmData".partData[7],
                           DataDelete => #tempDeleteData);
   IF #tempDeleteData THEN "Unit1.EmData".partData[4] := #ClearData; END_IF;
END_REGION

REGION Network 95: Transfer And Generate Hot Press Right To Transfer P&P Left [Em7 → Em5]
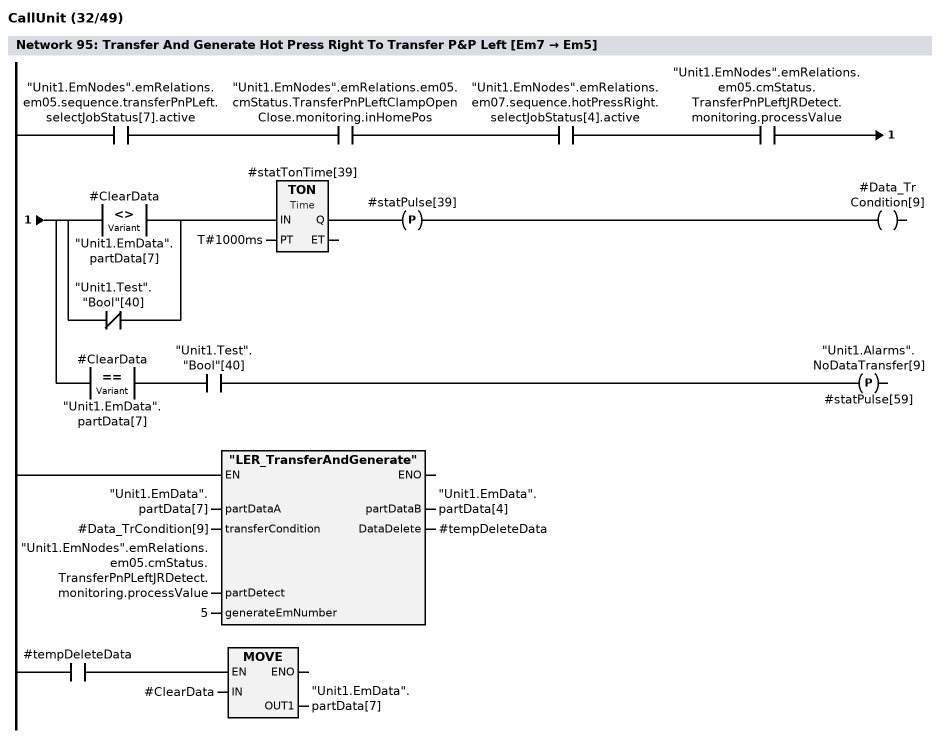
   #_w1 := "Unit1.EmNodes".emRelations.em05.sequence.transferPnPLeft.selectJobStatus[7].active AND "Unit1.EmNodes".emRelations.em05.cmStatus.TransferPnPLeftClampOpenClose.monitoring.inHomePos AND "Unit1.EmNodes".emRelations.em07.sequence.hotPressRight.selectJobStatus[4].active AND "Unit1.EmNodes".emRelations.em05.cmStatus.TransferPnPLeftJRDetect.monitoring.processValue;
   #statTonTime[39].TON(IN := #_w1 AND ((#ClearData <> "Unit1.EmData".partData[7]) OR NOT "Unit1.Test"."Bool"[40]),
                        PT := T#1000ms);
   #_w2 := #statTonTime[39].Q AND NOT #statPulse[39];   // rising edge
   #statPulse[39] := #statTonTime[39].Q;
   #Data_TrCondition[9] := #_w2;
   #_w3 := #_w1 AND (#ClearData = "Unit1.EmData".partData[7]) AND "Unit1.Test"."Bool"[40];
   "Unit1.Alarms".NoDataTransfer[9] := #_w3 AND NOT #statPulse[59];   // rising edge
   #statPulse[59] := #_w3;
   "LER_TransferAndGenerate"(partDataA := "Unit1.EmData".partData[7],
                           transferCondition := #Data_TrCondition[9],
                           partDetect := "Unit1.EmNodes".emRelations.em05.cmStatus.TransferPnPLeftJRDetect.monitoring.processValue,
                           generateEmNumber := 5,
                           partDataB => "Unit1.EmData".partData[4],
                           DataDelete => #tempDeleteData);
   IF #tempDeleteData THEN "Unit1.EmData".partData[7] := #ClearData; END_IF;
END_REGION

REGION Network 96: Transfer And Generate Transfer P&P Left To Hipot & Thickness [Em5 → Em8]
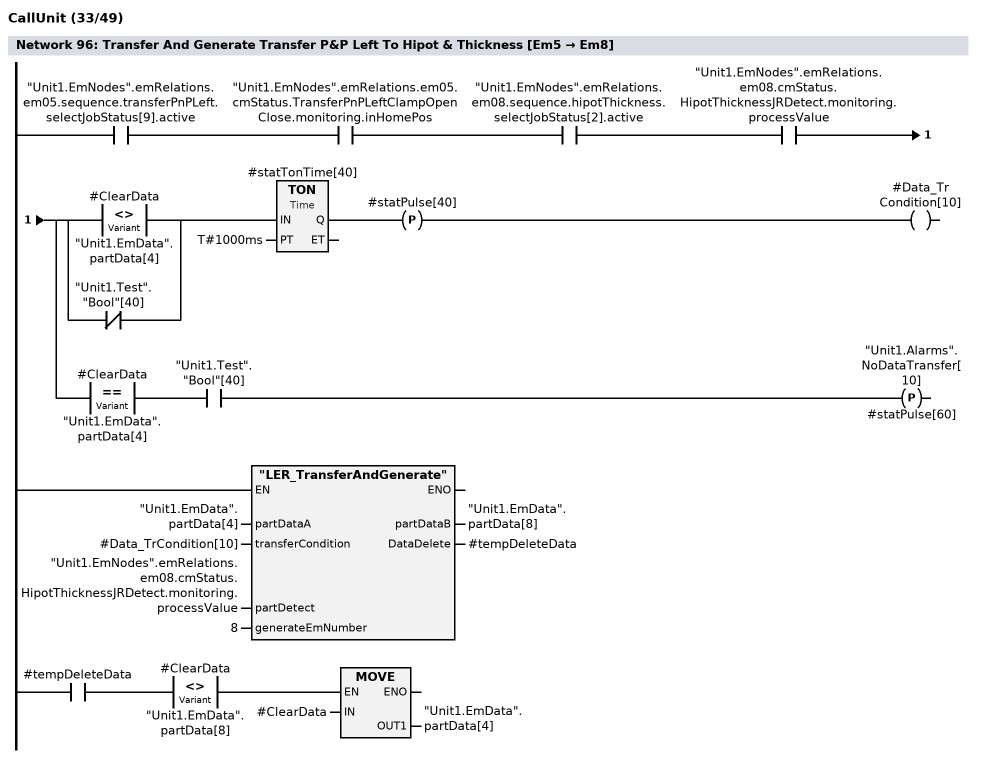
   #_w1 := "Unit1.EmNodes".emRelations.em05.sequence.transferPnPLeft.selectJobStatus[9].active AND "Unit1.EmNodes".emRelations.em05.cmStatus.TransferPnPLeftClampOpenClose.monitoring.inHomePos AND "Unit1.EmNodes".emRelations.em08.sequence.hipotThickness.selectJobStatus[2].active AND "Unit1.EmNodes".emRelations.em08.cmStatus.HipotThicknessJRDetect.monitoring.processValue;
   #statTonTime[40].TON(IN := #_w1 AND ((#ClearData <> "Unit1.EmData".partData[4]) OR NOT "Unit1.Test"."Bool"[40]),
                        PT := T#1000ms);
   #_w2 := #statTonTime[40].Q AND NOT #statPulse[40];   // rising edge
   #statPulse[40] := #statTonTime[40].Q;
   #Data_TrCondition[10] := #_w2;
   #_w3 := #_w1 AND (#ClearData = "Unit1.EmData".partData[4]) AND "Unit1.Test"."Bool"[40];
   "Unit1.Alarms".NoDataTransfer[10] := #_w3 AND NOT #statPulse[60];   // rising edge
   #statPulse[60] := #_w3;
   "LER_TransferAndGenerate"(partDataA := "Unit1.EmData".partData[4],
                           transferCondition := #Data_TrCondition[10],
                           partDetect := "Unit1.EmNodes".emRelations.em08.cmStatus.HipotThicknessJRDetect.monitoring.processValue,
                           generateEmNumber := 8,
                           partDataB => "Unit1.EmData".partData[8],
                           DataDelete => #tempDeleteData);
   IF #tempDeleteData AND (#ClearData <> "Unit1.EmData".partData[8]) THEN
       "Unit1.EmData".partData[4] := #ClearData;
   END_IF;
END_REGION

REGION Network 97: Transfer And Generate Hipot & Thickness To Transfer P&P Right [Em8 → Em5]
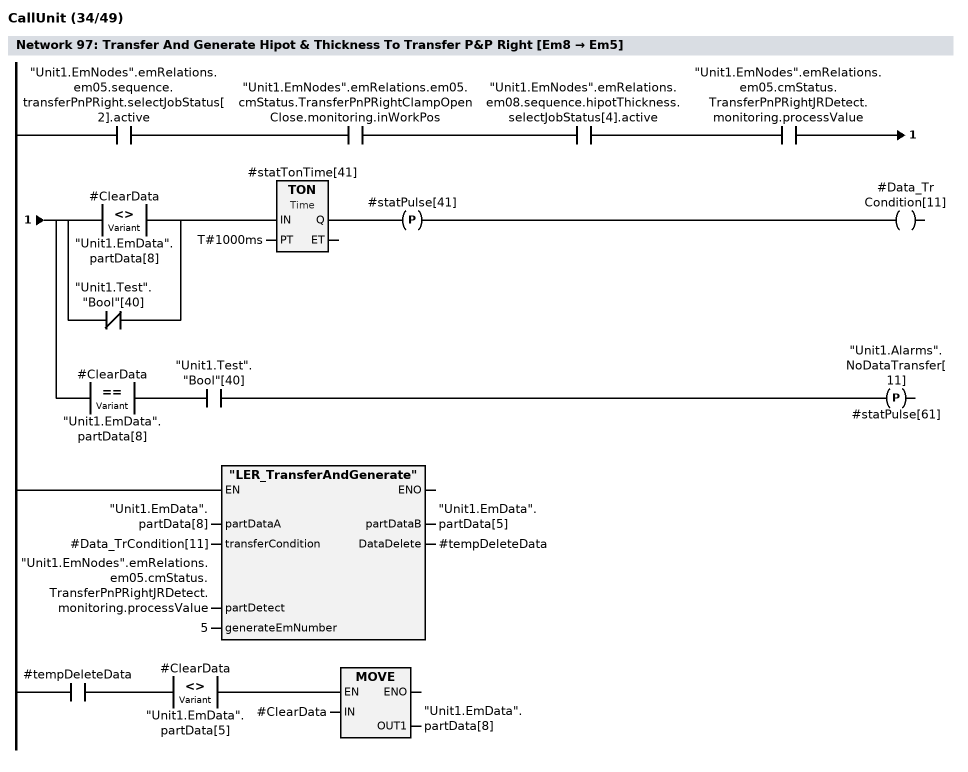
   #_w1 := "Unit1.EmNodes".emRelations.em05.sequence.transferPnPRight.selectJobStatus[2].active AND "Unit1.EmNodes".emRelations.em05.cmStatus.TransferPnPRightClampOpenClose.monitoring.inWorkPos AND "Unit1.EmNodes".emRelations.em08.sequence.hipotThickness.selectJobStatus[4].active AND "Unit1.EmNodes".emRelations.em05.cmStatus.TransferPnPRightJRDetect.monitoring.processValue;
   #statTonTime[41].TON(IN := #_w1 AND ((#ClearData <> "Unit1.EmData".partData[8]) OR NOT "Unit1.Test"."Bool"[40]),
                        PT := T#1000ms);
   #_w2 := #statTonTime[41].Q AND NOT #statPulse[41];   // rising edge
   #statPulse[41] := #statTonTime[41].Q;
   #Data_TrCondition[11] := #_w2;
   #_w3 := #_w1 AND (#ClearData = "Unit1.EmData".partData[8]) AND "Unit1.Test"."Bool"[40];
   "Unit1.Alarms".NoDataTransfer[11] := #_w3 AND NOT #statPulse[61];   // rising edge
   #statPulse[61] := #_w3;
   "LER_TransferAndGenerate"(partDataA := "Unit1.EmData".partData[8],
                           transferCondition := #Data_TrCondition[11],
                           partDetect := "Unit1.EmNodes".emRelations.em05.cmStatus.TransferPnPRightJRDetect.monitoring.processValue,
                           generateEmNumber := 5,
                           partDataB => "Unit1.EmData".partData[5],
                           DataDelete => #tempDeleteData);
   IF #tempDeleteData AND (#ClearData <> "Unit1.EmData".partData[5]) THEN
       "Unit1.EmData".partData[8] := #ClearData;
   END_IF;
END_REGION

REGION Network 98: Transfer And Generate Transfer P&P Right To Vision [Em5 → Em9]
